Yaskawa INFORM job: SKRZYNIA_5340_0_STOPNI_2OBR.JBI

/JOB
//NAME SKRZYNIA_5340_0_STOPNI_2OBR
///FOLDERNAME 02-SKRZYNIE_JOBS
//POS
///NPOS 607,607,0,50,0,0
///TOOL 0
///POSTYPE PULSE
///PULSE
C00000=1055,-24125,84372,288,19725,204
C00001=0,-15438,65714,0,-68532,0
C00002=4718,-16587,59952,3396,-65485,-935
C00003=32997,-21499,42555,27623,-61436,21376
C00004=31759,-20688,42932,26837,-60850,21559
C00005=28987,-21156,42712,24818,-60442,22222
C00006=33447,-21964,42352,27886,-61721,21330
C00007=37687,-23357,41794,30651,-63289,20620
C00008=38979,-19018,48057,32961,-64962,20678
C00009=37261,-18075,48526,31902,-64209,20901
C00010=35830,-17198,48994,31015,-63571,21092
C00011=34080,-17614,48768,29780,-63290,21485
C00012=37261,-18075,48526,31902,-64209,20901
C00013=47373,-21912,40596,41149,-66086,26950
C00014=45033,-20851,41104,39798,-65001,27223
C00015=42790,-19693,41704,38494,-63946,27495
C00016=41070,-20182,41442,37324,-63566,27891
C00017=45033,-20851,41104,39798,-65001,27223
C00018=45033,-20851,41104,39798,-65001,27223
C00019=59624,-29540,14278,64846,-60867,16042
C00020=57357,-28542,14780,63940,-59509,16120
C00021=56188,-29140,14476,63237,-58995,16387
C00022=59588,-29370,14363,64862,-60819,16012
C00023=62924,-29779,15793,65870,-63073,16252
C00024=59724,-28781,16276,64511,-61238,16415
C00025=57764,-27936,16704,63709,-60078,16488
C00026=56408,-28589,16373,62897,-59486,16787
C00027=59724,-28781,16276,64511,-61238,16415
C00028=87562,-48087,-13810,78020,-75252,11220
C00029=10104,-46603,4759,11228,-37390,-5046
C00030=0,-52280,40443,0,6876,0
C00031=1529,-42140,58025,-5964,2417,3265
C00032=0,-38374,23626,-1605,-51738,268
C00033=45044,-23015,37260,35797,-71879,25522
C00034=39973,-29571,18873,35060,-63052,24165
C00035=38620,-28701,19269,34339,-62304,24363
C00036=36409,-29254,19014,32896,-61805,24958
C00037=44451,-29039,21934,37281,-65892,23702
C00038=49472,-39353,6917,53118,-50908,20251
C00039=45058,-39356,3832,51653,-47640,20099
C00040=42883,-38319,4163,50577,-46309,20295
C00041=40255,-38926,3967,48502,-45334,21060
C00042=46774,-39679,3737,52663,-48537,19827
C00043=48708,-40455,3517,53615,-49689,19657
C00044=43798,-39237,3871,50850,-47027,20335
C00045=41951,-38324,4161,49930,-45891,20507
C00046=39836,-38844,3994,48234,-45126,21137
C00047=48489,-40338,3551,53521,-49551,19665
C00048=48489,-40338,3551,53521,-49551,19665
C00049=44432,-39026,3936,51363,-47247,20139
C00050=42487,-38069,4248,50403,-46050,20315
C00051=39061,-38795,4009,47695,-44769,21310
C00052=44432,-39026,3936,51363,-47247,20139
C00053=45358,-49480,-3557,50155,-49322,21260
C00054=1817,-44984,2816,-3462,-45659,1296
C00055=1445,-28771,30219,-502,-63201,-220
C00056=1148,-56354,34370,-22,3827,-10
C00057=0,-52280,40443,0,6876,0
C00058=0,-49898,44897,0,-65513,0
C00059=52002,-27630,35066,40617,-70496,28619
C00060=38179,-24916,32897,32855,-63545,30206
C00061=36484,-23889,33369,31863,-62698,30449
C00062=33804,-24434,33113,30025,-62179,31112
C00063=38179,-24916,32897,32855,-63545,30206
C00064=78369,-41260,16071,67181,-65880,21417
C00065=137,-45861,52341,97,-67596,-14
C00066=-31499,-58302,-23356,15027,12889,-13082
C00067=-52768,-43016,-26078,18373,38595,-18774
C00068=-89470,-32103,-32973,29905,69139,-31512
C00069=-68838,-26884,-24872,16972,64732,-23076
C00070=-53036,-11528,-12218,12363,64665,-17409
C00071=-51536,-9474,-10276,11905,64649,-16876
C00072=-51739,-9114,-7787,12104,63269,-17104
C00073=-53036,-11528,-12218,12363,64665,-17409
C00074=-17541,-26226,-24397,927,59032,-5038
C00075=-17541,-26226,-24397,927,59032,-5038
C00076=-16950,-23991,-22741,715,59568,-4818
C00077=-17036,-23563,-20101,755,58071,-4857
C00078=-17541,-26226,-24397,927,59032,-5038
C00079=34102,-23192,-21614,-15638,64271,13209
C00080=33423,-21885,-20599,-15423,64418,12942
C00081=32426,-19856,-18975,-15106,64629,12551
C00082=32578,-19611,-17013,-15290,63535,12762
C00083=33423,-21885,-20599,-15423,64418,12942
C00084=59339,-6070,-6417,-20979,72191,20891
C00085=59339,-6070,-6417,-20979,72191,20891
C00086=57897,-4256,-4562,-20702,71913,20431
C00087=58108,-3992,-2506,-20878,70835,20713
C00088=59339,-6070,-6417,-20979,72191,20891
C00089=42744,-35904,-30225,-18322,62562,16651
C00090=-53036,-11528,-12218,12363,64665,-17409
C00091=-77982,-26538,-29134,27151,66629,-27745
C00092=-70983,-8594,-1966,26503,59809,-49670
C00093=-80152,19776,40785,37351,72704,-50428
C00094=-79984,20154,42529,37516,71911,-50638
C00095=-79233,18397,40079,37458,71885,-50340
C00096=-79984,20154,42529,37516,71911,-50638
C00097=-73519,23289,38838,28890,77081,-45618
C00098=-73519,24511,42682,29072,75582,-46027
C00099=-73519,23289,38838,28890,77081,-45618
C00100=-88897,15706,42282,50101,71325,-56974
C00101=-88897,15706,42282,50101,71325,-56974
C00102=-87612,12343,37838,50071,70996,-56519
C00103=-85283,14202,40272,50301,69633,-56165
C00104=-87338,12550,38107,50098,70839,-56476
C00105=-84952,-1789,13569,34660,47724,-58955
C00106=-67641,-1674,11109,10330,44856,-44725
C00107=-66443,961,13975,9688,44721,-44210
C00108=-67641,-1674,11109,10330,44856,-44725
C00109=-67641,-376,15347,10694,42950,-44967
C00110=-67641,-1674,11109,10330,44856,-44725
C00111=-79040,417,20398,15965,28992,-57786
C00112=-76655,5212,30978,15501,25024,-57306
C00113=-76655,6949,35816,16758,23084,-57955
C00114=-76655,5212,30978,15501,25024,-57306
C00115=-74761,6919,33010,13466,24593,-56049
C00116=-80460,-2874,12270,15804,32253,-57809
C00117=-61258,-29124,-13156,26560,43617,-22150
C00118=-30420,-40507,-29240,27153,53235,15188
C00119=-18589,-38725,-21450,23338,47896,18931
C00120=-17722,-35233,-16455,23322,46926,19051
C00121=-17722,-33749,-12435,23948,45421,18620
C00122=-17722,-33892,-12819,23887,45564,18661
C00123=-16677,-31133,-11209,23138,46167,19311
C00124=-17819,-35820,-17540,23246,47228,19090
C00125=-74104,-11494,-6266,31916,75042,4269
C00126=-71226,-7329,2631,32115,71468,4273
C00127=-71226,-6504,5446,32343,70365,3922
C00128=-71226,-6611,5086,32313,70505,3967
C00129=-68386,-4058,7675,32040,69573,4789
C00130=-73314,-9412,-353,32206,72648,3829
C00131=51751,-31069,-22965,-10739,49070,48663
C00132=49028,-23852,-11575,-9841,46366,47823
C00133=49028,-23004,-8935,-10039,45204,47956
C00134=49028,-23118,-9286,-10013,45357,47939
C00135=47000,-20813,-7527,-8928,45644,47024
C00136=50476,-26208,-15307,-10408,47325,48332
C00137=90602,-5375,6902,-38786,69848,59444
C00138=83174,19950,50269,-44999,67580,58220
C00139=82362,17902,47383,-44926,67511,57879
C00140=83515,19072,48341,-44798,68200,58056
C00141=78091,19382,40247,-36371,72286,52960
C00142=78091,20664,44011,-36670,70997,53443
C00143=78091,19382,40247,-36371,72286,52960
C00144=88699,7296,38566,-55615,63182,60372
C00145=86803,3068,32674,-55410,62638,59657
C00146=84852,4315,34115,-55564,61561,59330
C00147=86803,3068,32674,-55410,62638,59657
C00148=92770,-2803,21719,-53893,67577,59421
C00149=73393,-10627,10934,-27897,30744,62458
C00150=70789,-6606,18800,-27824,27830,62140
C00151=69654,-4593,20814,-26755,27596,61444
C00152=70789,-6606,18800,-27824,27830,62140
C00153=70789,-5070,23059,-29482,26284,63017
C00154=70789,-6606,18800,-27824,27830,62140
C00155=83486,-8736,6503,-27040,35338,66550
C00156=77831,-2041,26192,-25270,18452,68895
C00157=77967,1961,32070,-26860,17569,69698
C00158=77967,5243,40752,-32914,14549,72656
C00159=77967,1961,32070,-26860,17569,69698
C00160=74560,4730,35257,-21622,16551,66717
C00161=77967,1961,32070,-26860,17569,69698
C00162=81109,-22356,2664,-22493,33121,60116
C00163=86168,-49730,-13668,-23926,46819,49343
C00164=44183,-52048,-7537,-24795,46064,51426
C00165=0,-52280,40443,0,6876,0
C00166=0,-52280,40443,0,6876,0
C00167=33629,-57276,-6399,46271,-24969,-2804
C00168=75493,-63502,-64712,103874,-64610,-6298
C00169=47446,-58597,-62761,109790,-45856,-10712
C00170=43673,-60069,-65334,114064,-43025,-9215
C00171=55379,-67378,-68041,108237,-48773,-4935
C00172=62671,-64213,-64640,104431,-56093,-7372
C00173=28458,-50318,6850,47420,-25887,-3347
C00174=0,-52280,40443,0,6876,0
C00175=1055,-24125,84372,288,19725,204
C00176=0,-15438,65714,0,-68532,0
C00177=0,-15438,65714,966,-70097,42926
C00178=69988,-9219,57065,61610,-82752,27767
C00179=63113,-6157,59685,58080,-79692,28271
C00180=46309,-5455,68070,40267,-75151,29719
C00181=49471,-5188,67710,43421,-76082,29577
C00182=63113,-6157,59685,58080,-79692,28271
C00183=69988,-9219,57065,61610,-82752,27767
C00184=0,-15438,65714,966,-70097,42926
C00185=0,-15438,65714,0,-68532,0
C00186=1055,-24125,84372,288,19725,204
C00187=1055,-24125,84372,288,19725,204
C00188=0,-52280,40443,0,6876,0
C00189=0,-17525,61946,0,273,32004
C00190=54446,-4421,37881,-48560,57645,57448
C00191=45059,-5790,38757,-53071,45868,54447
C00192=47306,-4859,57027,-85859,41058,71744
C00193=46362,-329,57203,-69834,42671,59860
C00194=35194,-2896,34959,-39493,48020,38101
C00195=43067,2853,36106,-38598,60324,43004
C00196=45059,-5790,38757,-53071,45868,54447
C00197=54446,-4421,37881,-48560,57645,57448
C00198=0,-17525,61946,0,273,32004
C00199=0,-52280,40443,0,6876,0
C00200=0,-52280,40443,0,6876,0
C00201=0,-52280,40443,0,6876,0
C00202=0,-52280,40443,0,-42737,40640
C00203=0,-52280,40443,0,-42737,40640
C00204=64551,-35409,28076,75550,-44539,17239
C00205=49799,-25338,45366,61341,-39751,21495
C00206=45731,-22710,35392,68644,-36821,18294
C00207=38151,-27944,23982,59630,-35957,20215
C00208=38219,-25330,29845,57337,-37014,21581
C00209=43117,-27612,29118,67655,-35359,18183
C00210=39863,-22026,47404,54615,-35502,22403
C00211=0,-52277,40442,0,6872,2
C00212=0,-38538,66749,0,-898,0
C00213=0,-52280,40443,0,-79033,35417
C00214=46775,-35113,22190,42926,-67531,20697
C00215=52587,-26056,25345,47610,-66542,17970
C00216=46075,-25504,24484,44216,-63256,18807
C00217=46254,-27712,19552,44922,-62123,18131
C00218=53914,-29436,22058,48262,-67266,17843
C00219=46775,-35113,22190,42926,-67531,20697
C00220=0,-52280,40443,0,-79033,35417
C00221=0,-52280,40443,0,-61239,28081
C00222=53819,-14110,13758,-46164,60155,50576
C00223=48398,-14119,9451,-44868,59619,48162
C00224=41013,-18640,20407,-60592,39621,52880
C00225=26504,-16872,16016,-34457,37392,33859
C00226=48398,-14119,9451,-44868,59619,48162
C00227=53819,-14110,13758,-46164,60155,50576
C00228=0,-52280,40443,0,-61239,28081
C00229=404,-42897,57020,-1574,2523,869
C00230=404,-42897,57020,-1574,2523,869
C00231=0,-52280,40443,0,6876,0
C00232=-99253,-13690,44082,59847,13407,-31313
C00233=-87814,-12734,20141,45739,-14352,-64418
C00234=-86669,-6582,30812,41148,-16781,-62025
C00235=-85055,-5827,31548,44003,-17420,-63187
C00236=-85971,-6262,31124,42409,-17052,-62539
C00237=-86650,-5303,32069,41395,-16716,-62141
C00238=-94954,-14494,-1860,-7818,15857,-59130
C00239=-94513,13660,61459,-3970,3134,-58997
C00240=-94981,20459,77123,-7495,-2517,-57346
C00241=-85971,-6262,31124,42409,-17052,-62539
C00242=-86125,-12470,22545,29004,-25567,-58412
C00243=-83883,-11340,22525,32952,-25567,-60136
C00244=-82768,-10824,22986,34487,-25904,-60776
C00245=-83883,-11340,22525,32952,-25567,-60136
C00246=-85143,-9772,23941,31487,-24966,-59556
C00247=-83883,-11340,22525,32952,-25567,-60136
C00248=-85732,-21202,11427,30682,-24763,-59235
C00249=-84150,-10929,23786,31981,-25941,-59678
C00250=-83036,-10419,24246,33504,-26268,-60308
C00251=-84150,-10929,23786,31981,-25941,-59678
C00252=-85291,-9507,25078,30650,-25411,-59154
C00253=-84150,-10929,23786,31981,-25941,-59678
C00254=-85786,-16909,14677,31743,-23900,-59790
C00255=-84150,-10498,24888,31517,-26306,-59436
C00256=-83174,-10052,25293,32841,-26587,-59984
C00257=-84150,-10498,24888,31517,-26306,-59436
C00258=-85258,-9112,26156,30226,-25800,-58928
C00259=-84150,-10498,24888,31517,-26306,-59436
C00260=-87841,-18519,13420,28367,-23534,-58339
C00261=-85040,-10859,24618,30253,-26091,-58908
C00262=-83241,-10052,25348,32714,-26598,-59924
C00263=-84150,-10465,24972,31484,-26336,-59417
C00264=-85145,-9228,26102,30329,-25881,-58963
C00265=-84150,-10465,24972,31484,-26336,-59417
C00266=-86371,-18277,13606,30568,-23951,-59265
C00267=-84345,-11688,21985,32461,-25312,-59957
C00268=-83211,-11173,22442,34044,-25650,-60618
C00269=-84345,-11688,21985,32461,-25312,-59957
C00270=-85283,-10526,23025,31366,-24861,-59525
C00271=-84345,-11688,21985,32461,-25312,-59957
C00272=-86191,-19647,12567,30467,-24278,-59187
C00273=-84345,-10877,24073,31552,-26006,-59481
C00274=-83051,-10286,24607,33321,-26381,-60213
C00275=-84345,-10877,24073,31552,-26006,-59481
C00276=-85179,-9842,25009,30582,-25619,-59100
C00277=-84345,-10877,24073,31552,-26006,-59481
C00278=-85438,-18022,14839,31140,-24818,-59429
C00279=-84247,-11820,22550,32049,-25753,-59727
C00280=-84104,-10976,23642,32111,-25899,-59738
C00281=-82990,-10465,24105,33639,-26227,-60372
C00282=-84104,-10976,23642,32111,-25899,-59738
C00283=-84898,-9998,24525,31196,-25529,-59378
C00284=-84104,-10976,23642,32111,-25899,-59738
C00285=-86610,-16845,14732,30573,-23614,-59301
C00286=-84104,-10864,23927,31990,-25993,-59674
C00287=-82824,-10273,24459,33737,-26370,-60397
C00288=-84104,-10864,23927,31990,-25993,-59674
C00289=-84789,-10021,24690,31200,-25673,-59363
C00290=-84104,-10864,23927,31990,-25993,-59674
C00291=-83806,-19585,12613,33764,-25080,-60559
C00292=-83924,-10205,25475,31619,-26533,-59453
C00293=-82780,-9675,25960,33156,-26866,-60087
C00294=-83924,-10205,25475,31619,-26533,-59453
C00295=-84478,-9530,26093,30986,-26280,-59206
C00296=-83924,-10205,25475,31619,-26533,-59453
C00297=-87149,-17993,13826,29513,-23647,-58830
C00298=-84920,-13182,20975,31162,-25481,-59361
C00299=-83711,-10572,24852,32056,-26475,-59649
C00300=-82779,-10142,25241,33309,-26748,-60166
C00301=-83711,-10572,24852,32056,-26475,-59649
C00302=-84370,-9774,25579,31305,-26170,-59356
C00303=-83711,-10572,24852,32056,-26475,-59649
C00304=-83642,-3679,42021,23358,-36761,-56118
C00305=-85886,-5975,41264,18964,-40261,-54782
C00306=-83919,-11632,22322,32811,-25616,-60079
C00307=-82884,-11162,22742,34234,-25925,-60671
C00308=-83919,-11632,22322,32811,-25616,-60079
C00309=-84723,-10654,23196,31887,-25230,-59715
C00310=-83919,-11632,22322,32811,-25616,-60079
C00311=-87348,-16035,7353,17528,-35245,-56477
C00312=-86244,-15062,8172,18754,-35315,-57058
C00313=-86244,-16649,3638,19674,-33501,-57585
C00314=-85308,-16228,3988,20718,-33648,-58082
C00315=-86244,-16649,3638,19674,-33501,-57585
C00316=-86740,-15973,4201,19194,-33277,-57362
C00317=-86244,-16649,3638,19674,-33501,-57585
C00318=-73780,-8639,20128,34258,-51705,-52097
C00319=-90711,-17528,-28778,11328,-28245,-57111
C00320=-92565,-19610,-33223,7138,-24591,-57051
C00321=-91512,-19116,-32812,8551,-24603,-57834
C00322=-92565,-19610,-33223,7138,-24591,-57051
C00323=-93003,-18716,-32476,6600,-24397,-56752
C00324=-92565,-19610,-33223,7138,-24591,-57051
C00325=-92565,-19610,-33223,7138,-24591,-57051
C00326=-95836,-54375,-51122,6031,-17685,-48210
C00327=-95836,-54375,-51122,6031,-17685,-48210
C00328=-43821,-47238,-2775,-3022,56549,-3681
C00329=-20126,-26882,59542,2406,16879,-9162
C00330=-20126,-26882,59542,2406,16879,-9162
C00331=98601,-10520,92678,4674,-40855,-9615
C00332=95537,-19831,-2695,-2933,-44471,35837
C00333=92548,-20391,-28429,-6186,-30623,55200
C00334=91429,-17018,-28974,-8057,-27827,56250
C00335=91429,-17018,-28974,-8057,-27827,56250
C00336=90371,-16495,-28521,-9286,-27856,56953
C00337=91429,-17018,-28974,-8057,-27827,56250
C00338=92033,-15799,-27911,-7415,-27588,55880
C00339=91429,-17018,-28974,-8057,-27827,56250
C00340=92548,-20391,-28429,-6186,-30623,55200
C00341=91156,-15018,-4648,-8036,-38181,54813
C00342=90585,-14766,-4428,-8565,-38201,55100
C00343=88830,-13959,-3717,-10186,-38284,55977
C00344=89897,-14456,-4157,-9202,-38230,55445
C00345=90761,-12944,-2809,-8452,-37927,55043
C00346=89897,-14456,-4157,-9202,-38230,55445
C00347=89910,-11217,67535,-9455,-58896,55399
C00348=89910,-11217,67535,-9455,-58896,55399
C00349=85786,-16735,14816,-31782,-23869,59812
C00350=83514,-12996,17929,-35760,-24132,61552
C00351=82251,-12406,18443,-37550,-24551,62308
C00352=83514,-12996,17929,-35760,-24132,61552
C00353=84258,-12095,18717,-34917,-23742,61217
C00354=83514,-12996,17929,-35760,-24132,61552
C00355=87149,-17993,13826,-29513,-23647,58830
C00356=83118,-12818,18089,-36330,-24263,61791
C00357=81915,-12248,18589,-38020,-24666,62504
C00358=83118,-12818,18089,-36330,-24263,61791
C00359=83897,-11882,18912,-35460,-23856,61445
C00360=83118,-12818,18089,-36330,-24263,61791
C00361=83806,-19585,12613,-33764,-25080,60559
C00362=82998,-13006,17925,-36445,-24332,61826
C00363=81675,-12378,18472,-38297,-24777,62607
C00364=82998,-13006,17925,-36445,-24332,61826
C00365=83876,-11958,18841,-35466,-23874,61442
C00366=82998,-13006,17925,-36445,-24332,61826
C00367=86610,-16845,14732,-30573,-23614,59301
C00368=82493,-13239,17725,-37070,-24559,62089
C00369=81406,-12724,18174,-38578,-24928,62723
C00370=82493,-13239,17725,-37070,-24559,62089
C00371=83436,-12134,18690,-36041,-24064,61684
C00372=82493,-13239,17725,-37070,-24559,62089
C00373=84814,-16043,15376,-33312,-24093,60464
C00374=82555,-13613,17404,-36910,-24580,62015
C00375=81384,-13062,17878,-38534,-24974,62698
C00376=82555,-13613,17404,-36910,-24580,62015
C00377=83566,-12434,18427,-35805,-24047,61580
C00378=82555,-13613,17404,-36910,-24580,62015
C00379=86191,-19647,12567,-30467,-24278,59187
C00380=82500,-13648,17375,-36975,-24607,62039
C00381=81467,-13161,17792,-38413,-24955,62645
C00382=82500,-13648,17375,-36975,-24607,62039
C00383=83481,-12505,18364,-35905,-24087,61617
C00384=82500,-13648,17375,-36975,-24607,62039
C00385=86371,-18277,13606,-30568,-23951,59265
C00386=82904,-13790,17251,-36416,-24470,61808
C00387=81715,-13237,17726,-38081,-24865,62509
C00388=82904,-13790,17251,-36416,-24470,61808
C00389=83686,-12878,18037,-35556,-24055,61469
C00390=82904,-13790,17251,-36416,-24470,61808
C00391=87841,-18519,13420,-28367,-23534,58339
C00392=82748,-13879,17174,-36603,-24542,61883
C00393=81692,-13388,17594,-38077,-24893,62505
C00394=82748,-13879,17174,-36603,-24542,61883
C00395=83607,-12881,18032,-35663,-24082,61515
C00396=82748,-13879,17174,-36603,-24542,61883
C00397=85786,-16909,14677,-31743,-23900,59790
C00398=82520,-14198,16902,-36833,-24674,61972
C00399=81460,-13708,17319,-38301,-25026,62591
C00400=82520,-14198,16902,-36833,-24674,61972
C00401=83571,-12989,17938,-35691,-24113,61524
C00402=82520,-14198,16902,-36833,-24674,61972
C00403=85732,-21202,11427,-30682,-24763,59235
C00404=82398,-14365,16763,-36952,-24745,62014
C00405=81172,-13798,17245,-38643,-25153,62725
C00406=82398,-14365,16763,-36952,-24745,62014
C00407=83600,-12984,17944,-35650,-24102,61504
C00408=82398,-14365,16763,-36952,-24745,62014
C00409=92346,-18713,13565,-21110,-22545,55257
C00410=82794,-13980,17083,-36511,-24538,61844
C00411=81518,-13384,17592,-38292,-24965,62594
C00412=82794,-13980,17083,-36511,-24538,61844
C00413=83714,-12912,18003,-35501,-24048,61445
C00414=82794,-13980,17083,-36511,-24538,61844
C00415=86140,-12802,12665,-93523,-10743,85795
C00416=86140,-12802,12665,-93523,-10743,85795
C00417=85030,-12289,13120,-93723,-11463,85776
C00418=86140,-12802,12665,-93523,-10743,85795
C00419=86958,-11660,13681,-94506,-10238,86349
C00420=86140,-12802,12665,-93523,-10743,85795
C00421=86625,-13020,12474,-93432,-10428,85802
C00422=86720,-13063,12436,-93414,-10366,85804
C00423=85672,-12588,12853,-93609,-11048,85787
C00424=86091,-12781,12683,-93534,-10775,85794
C00425=86978,-11540,13790,-94601,-10225,86395
C00426=86091,-12781,12683,-93534,-10775,85794
C00427=86674,107,23869,25042,24033,51593
C00428=86674,107,23869,25042,24033,51593
C00429=86674,1750,28532,27061,22272,50559
C00430=86674,107,23869,25042,24033,51593
C00431=86830,-21199,-17039,14859,33768,55796
C00432=85045,-36869,-4353,-28502,-22832,52282
C00433=0,-24029,84339,0,19981,0
C00434=0,-24029,84339,0,19981,0
C00435=3172,-24246,80980,3465,15913,689
C00436=-86563,-26985,13879,10257,-21548,-45530
C00437=-86191,-19647,12567,30467,-24278,-59187
C00438=-83221,-13587,17636,37793,-25116,-62228
C00439=-91978,-13833,14560,12391,-18633,-51524
C00440=-94992,-13830,14285,1276,-18012,-46664
C00441=-84074,-17488,11256,38660,-23649,-62784
C00442=-73679,-33270,1000,44272,-31600,-64253
C00443=-86926,-60758,23267,6576,1160,-9545
C00444=0,-52280,40443,0,6876,0
C00445=82475,-58079,26734,835,4084,4444
C00446=97932,-26840,7691,8784,-23444,42538
C00447=87166,-16607,16322,-25365,-24201,56345
C00448=84699,-11354,21752,-29145,-24735,57949
C00449=84804,-11023,22730,-28561,-25071,57659
C00450=85100,-26994,10417,-24982,-28140,55821
C00451=0,-52280,40443,0,6876,0
C00452=0,-52280,40443,0,6876,0
C00453=-90140,-60305,18108,-2708,1721,-7625
C00454=-95594,-27428,6866,-4663,-19832,-42154
C00455=-98688,-13767,16447,-18366,-10080,-35766
C00456=-98964,-4977,31041,-27811,-8682,-30400
C00457=-98987,-3006,34487,-29035,-8628,-29652
C00458=-99668,3923,47993,-36046,-8554,-25749
C00459=-97898,6199,51529,-29419,-5862,-29460
C00460=-93331,7027,46084,-21637,6926,-34654
C00461=-93331,9643,52589,-32935,4701,-29330
C00462=-91881,12566,59903,-8075,11651,-42601
C00463=-91392,18044,70719,-12774,8436,-40275
C00464=-95084,15513,53253,-335,18313,-46866
C00465=-99268,-13088,27343,-18620,-14105,-35021
C00466=-90140,-60305,18108,-2708,1721,-7625
C00467=0,-52280,40443,0,6876,0
C00468=84259,-57935,27522,-3761,3673,6310
C00469=86507,-39672,4297,-27618,-16640,46340
C00470=73669,-37119,-20783,-92053,-19719,85232
C00471=86539,-20830,1725,-71850,-11773,76853
C00472=94927,-16191,10904,-46169,-1414,61414
C00473=97704,-11547,13178,-56709,4181,66931
C00474=98708,-8628,11747,-16202,14842,48818
C00475=96432,-319,21323,-3495,24089,38404
C00476=97976,685,17732,-6153,31139,39163
C00477=96085,-4775,15361,-2075,25096,37900
C00478=101780,15887,17889,-10773,66834,38316
C00479=97846,5957,18050,-4866,41853,38411
C00480=100487,-9453,-1206,-10413,41328,41147
C00481=96250,-19428,-8283,-4838,27297,37910
C00482=86507,-39672,4297,-27618,-16640,46340
C00483=84259,-57935,27522,-3761,3673,6310
C00484=0,-52280,40443,0,6876,0
C00485=0,-27933,77061,0,20812,0
C00486=0,-27933,77061,0,20812,0
C00487=0,-52280,40443,0,6876,0
C00488=-91970,-60791,14435,-3343,512,-9412
C00489=-98647,-24138,10005,-11519,-21203,-39749
C00490=-99883,-13980,22886,-11640,-25090,-40341
C00491=-99702,-9154,61728,-1148,-61809,-40243
C00492=-84328,-13042,29707,23458,-33731,-54641
C00493=-83101,-4179,39208,25894,-34785,-55667
C00494=-82881,-4330,38692,26392,-34479,-55866
C00495=-76259,-18287,26646,31659,-38322,-57579
C00496=-89741,-28009,12101,4461,-28076,-46404
C00497=-91970,-60791,14435,-3343,512,-9412
C00498=0,-52280,40443,0,6876,0
C00499=91083,-60784,14823,-9043,-825,15173
C00500=83869,-19403,12921,-33769,-24740,60260
C00501=83869,-19403,12921,-33769,-24740,60260
C00502=83932,-19538,53415,-33663,-71112,60249
C00503=83932,-19538,53415,-33663,-71112,60249
C00504=82480,-12247,21118,-35440,-26416,60009
C00505=82194,-11433,19802,-37650,-25323,61125
C00506=81904,-9374,24711,-35791,-26879,60109
C00507=79790,-20261,14917,-36681,-28829,60258
C00508=76554,-29711,-1870,-46042,-25952,65654
C00509=91083,-60784,14823,-9043,-825,15173
C00510=0,-52280,40443,0,6876,0
C00511=-91526,-60598,16699,7584,176,-13289
C00512=-81382,-25890,9219,35455,-25500,-59095
C00513=-86453,-20958,12525,30076,-22568,-57089
C00514=-86589,-16097,16237,31250,-21582,-57704
C00515=-98933,-11298,20505,-13970,-18736,-37953
C00516=-98281,-10965,21163,-11559,-18548,-39330
C00517=-85424,-18472,14402,34409,-22969,-58895
C00518=-74746,-27148,8488,44263,-29128,-62418
C00519=-81326,-27507,8265,35533,-26282,-59001
C00520=-91415,-60262,16631,7870,-73,-13734
C00521=24,-24029,84339,7,19981,5
C00522=100404,-52373,45687,-1822,14816,-5144
C00523=75939,-26469,7919,-40869,-29645,63133
C00524=81882,-22565,10470,-35355,-26404,61107
C00525=82801,-12246,21732,-34208,-26055,60642
C00526=91844,-10818,23389,-8611,-22226,49798
C00527=96558,-9677,26191,5829,-23135,43648
C00528=77262,-23244,14300,-38922,-31295,61912
C00529=78410,-22868,15324,-38001,-30064,61274
C00530=96357,-33562,33410,58602,-23427,10353
C00531=568,-24029,84339,168,19981,112
C00532=-91970,-60791,14435,-3343,512,-9412
C00533=-98991,-22833,11519,-12824,-17638,-36336
C00534=-86376,-13627,18436,38326,-18406,-58533
C00535=-85581,-10814,20279,41280,-18093,-59893
C00536=-85551,-10406,21021,40925,-18257,-59713
C00537=-86274,-24518,9978,34497,-20333,-56613
C00538=-91684,-53777,2301,20525,-9313,-33684
C00539=-67305,-55044,34987,1504,5690,-2468
C00540=0,-52280,40443,0,6876,0
C00541=77036,-56616,31288,-2531,4707,4197
C00542=84359,-28321,8817,-32860,-20485,54199
C00543=81156,-16932,14874,-39538,-26422,62851
C00544=93122,-15135,13007,-5735,-18111,48773
C00545=90767,-14192,15510,-13532,-19632,52035
C00546=77970,-27630,4721,-41834,-28549,63607
C00547=81111,-35571,7141,-33980,-21909,52006
C00548=82626,-57814,28323,-4146,3364,6346
C00549=0,-52280,40443,0,6876,0
C00550=0,-28135,76691,0,20839,0
C00551=0,-28135,76691,0,20839,0
C00552=-45332,-39712,59352,-1730,18713,2903
C00553=-94065,-8316,59352,-1730,-37754,-40387
C00554=-100331,-14895,33931,-8215,-36518,-40227
C00555=-98931,-8578,39429,-6260,-48307,-43744
C00556=-100336,-4176,46216,-7600,-55875,-44633
C00557=-93952,8947,73671,995,-68520,-43850
C00558=-98791,-3170,32594,-4861,-60761,-43748
C00559=-98768,4156,37660,-4945,-58738,-43661
C00560=-98673,-12696,-17797,-7569,-33360,-41896
C00561=-99330,-14840,-29426,-9917,-27109,-40593
C00562=-99605,-15546,-21493,-8548,-33053,-41326
C00563=-100467,-8208,-2562,-8095,-44661,-42156
C00564=-93952,8947,73671,995,-68520,-43850
C00565=-88754,54,62805,4404,-67858,-45120
C00566=-100222,-4532,45667,-7492,-55263,-44561
C00567=-100331,-14895,33931,-8215,-36518,-40227
C00568=-94065,-8316,59352,-1730,-37754,-40387
C00569=-45544,-32973,71870,-2133,15168,3033
C00570=0,-28135,76691,0,20839,0
C00571=54178,-17846,77779,596,-29686,20997
C00572=54178,-17846,77779,596,-29686,20997
C00573=99462,-18987,75418,611,-28919,20989
C00574=98707,-9390,78674,1080,-71212,38250
C00575=98768,-5182,41096,1808,-44974,38308
C00576=100431,1771,51615,3823,-56746,39115
C00577=97953,-6621,17555,2289,-50176,39420
C00578=95834,-5353,18817,760,-50052,40242
C00579=86453,-3910,18511,-13431,-48443,44868
C00580=88887,-11110,-8515,-11527,-36861,46615
C00581=88808,-13839,-20865,-13699,-30585,47852
C00582=90457,-16080,-12990,-9972,-37305,45724
C00583=97953,-6621,17555,2289,-50176,39420
C00584=100431,1771,51615,3823,-56746,39115
C00585=98768,-5182,41096,1808,-44974,38308
C00586=98707,-9390,78674,1080,-71212,38250
C00587=0,-28135,76691,0,20839,0
C00588=0,-28135,76691,0,20839,0
C00589=-91526,-60598,16699,7584,176,-13289
C00590=-81382,-25890,9219,35455,-25500,-59095
C00591=-81382,-25890,9219,35455,-25500,-59095
C00592=-85509,-13950,19358,32213,-22393,-58041
C00593=-96341,-12086,19487,-5053,-17846,-42145
C00594=-97523,-9822,24708,-8570,-19966,-40659
C00595=-84656,-25369,12054,31249,-26195,-57129
C00596=-82652,-57346,29982,2770,3944,-5064
C00597=0,-52280,40443,0,6876,0
C00598=60653,-54633,35892,-1212,5841,2035
C00599=77942,-28227,6869,-38010,-29303,61907
C00600=82500,-13648,17375,-36975,-24607,62039
C00601=80731,-11587,18684,-41654,-25449,63953
C00602=80409,-10373,22284,-40214,-26848,63104
C00603=64389,-31987,5108,-50419,-37074,66126
C00604=60653,-54633,35892,-1212,5841,2035
C00605=0,-52280,40443,0,6876,0
C00606=0,-28167,76633,0,20843,0
BC00000=413138
BC00001=413138
BC00002=388163
BC00003=356740
BC00004=356740
BC00005=356740
BC00006=356740
BC00007=356740
BC00008=407176
BC00009=407176
BC00010=407176
BC00011=407176
BC00012=407176
BC00013=479433
BC00014=479433
BC00015=479433
BC00016=479433
BC00017=479433
BC00018=530237
BC00019=530237
BC00020=530237
BC00021=530237
BC00022=530237
BC00023=601977
BC00024=601977
BC00025=601977
BC00026=601977
BC00027=601977
BC00028=601977
BC00029=522422
BC00030=522422
BC00031=671734
BC00032=689202
BC00033=689202
BC00034=689202
BC00035=689202
BC00036=689202
BC00037=689202
BC00038=726463
BC00039=726463
BC00040=726463
BC00041=726463
BC00042=726463
BC00043=782137
BC00044=782137
BC00045=782137
BC00046=782137
BC00047=782137
BC00048=850421
BC00049=850421
BC00050=850421
BC00051=850421
BC00052=850421
BC00053=850421
BC00054=823841
BC00055=797607
BC00056=755227
BC00057=755227
BC00058=915219
BC00059=914226
BC00060=914226
BC00061=914226
BC00062=914226
BC00063=914226
BC00064=914226
BC00065=922367
BC00066=927819
BC00067=927819
BC00068=927819
BC00069=943180
BC00070=943180
BC00071=943180
BC00072=943180
BC00073=943180
BC00074=943180
BC00075=943180
BC00076=943180
BC00077=943180
BC00078=943180
BC00079=943180
BC00080=943180
BC00081=943180
BC00082=943180
BC00083=943180
BC00084=943180
BC00085=943180
BC00086=943180
BC00087=943180
BC00088=943180
BC00089=943180
BC00090=943180
BC00091=943180
BC00092=943180
BC00093=943180
BC00094=943182
BC00095=943182
BC00096=943182
BC00097=943182
BC00098=943182
BC00099=943182
BC00100=943182
BC00101=943182
BC00102=943182
BC00103=943182
BC00104=943182
BC00105=943182
BC00106=943182
BC00107=943182
BC00108=943182
BC00109=943182
BC00110=943182
BC00111=943182
BC00112=943182
BC00113=943182
BC00114=943182
BC00115=943182
BC00116=943182
BC00117=943183
BC00118=943184
BC00119=943184
BC00120=943184
BC00121=943184
BC00122=943184
BC00123=943184
BC00124=943184
BC00125=943184
BC00126=943184
BC00127=943184
BC00128=943184
BC00129=943156
BC00130=943170
BC00131=943170
BC00132=943170
BC00133=943170
BC00134=943170
BC00135=943170
BC00136=943170
BC00137=943184
BC00138=943184
BC00139=943184
BC00140=943184
BC00141=943184
BC00142=943184
BC00143=943184
BC00144=943184
BC00145=943184
BC00146=943184
BC00147=943184
BC00148=943184
BC00149=943184
BC00150=943184
BC00151=943184
BC00152=943184
BC00153=943184
BC00154=943184
BC00155=943184
BC00156=943184
BC00157=943184
BC00158=943184
BC00159=943184
BC00160=943184
BC00161=943184
BC00162=911399
BC00163=884954
BC00164=838173
BC00165=838173
BC00166=727925
BC00167=734552
BC00168=750834
BC00169=750837
BC00170=810605
BC00171=811927
BC00172=760768
BC00173=744267
BC00174=744267
BC00175=413138
BC00176=413138
BC00177=413138
BC00178=408626
BC00179=408626
BC00180=408753
BC00181=347392
BC00182=408626
BC00183=408626
BC00184=413138
BC00185=413138
BC00186=413138
BC00187=505502
BC00188=697681
BC00189=697681
BC00190=733666
BC00191=758324
BC00192=766520
BC00193=794510
BC00194=817294
BC00195=794510
BC00196=758324
BC00197=733666
BC00198=697681
BC00199=697681
BC00200=697681
BC00201=841681
BC00202=841681
BC00203=884227
BC00204=901088
BC00205=895224
BC00206=896289
BC00207=924873
BC00208=968077
BC00209=921975
BC00210=887634
BC00211=824879
BC00212=507816
BC00213=507816
BC00214=552804
BC00215=552804
BC00216=551170
BC00217=493239
BC00218=491979
BC00219=552804
BC00220=507816
BC00221=507816
BC00222=507816
BC00223=531288
BC00224=531293
BC00225=591068
BC00226=531288
BC00227=507816
BC00228=507816
BC00229=507816
BC00230=737809
BC00231=848972
BC00232=861901
BC00233=963633
BC00234=963633
BC00235=963633
BC00236=963633
BC00237=963633
BC00238=963633
BC00239=963633
BC00240=963633
BC00241=963633
BC00242=963633
BC00243=963633
BC00244=963633
BC00245=963633
BC00246=963633
BC00247=963633
BC00248=902188
BC00249=895372
BC00250=895372
BC00251=895372
BC00252=895372
BC00253=895372
BC00254=840744
BC00255=840744
BC00256=840744
BC00257=840744
BC00258=840744
BC00259=840744
BC00260=779300
BC00261=771332
BC00262=771332
BC00263=771332
BC00264=771332
BC00265=771332
BC00266=717855
BC00267=717855
BC00268=717855
BC00269=717855
BC00270=717855
BC00271=717855
BC00272=656405
BC00273=649173
BC00274=649173
BC00275=649173
BC00276=649173
BC00277=649173
BC00278=594961
BC00279=594961
BC00280=594961
BC00281=594961
BC00282=594961
BC00283=594961
BC00284=594961
BC00285=533517
BC00286=525229
BC00287=525229
BC00288=525229
BC00289=525229
BC00290=525229
BC00291=472073
BC00292=472073
BC00293=472073
BC00294=472073
BC00295=472073
BC00296=472073
BC00297=410629
BC00298=405662
BC00299=402968
BC00300=402968
BC00301=402968
BC00302=402968
BC00303=402968
BC00304=402968
BC00305=349186
BC00306=349186
BC00307=349186
BC00308=349186
BC00309=349186
BC00310=349186
BC00311=336469
BC00312=336469
BC00313=336469
BC00314=336469
BC00315=336469
BC00316=336469
BC00317=336469
BC00318=367602
BC00319=367601
BC00320=367601
BC00321=367601
BC00322=367601
BC00323=367601
BC00324=367601
BC00325=425303
BC00326=425303
BC00327=514953
BC00328=463119
BC00329=419862
BC00330=484962
BC00331=484962
BC00332=395463
BC00333=369502
BC00334=369502
BC00335=369502
BC00336=369502
BC00337=369502
BC00338=369502
BC00339=369502
BC00340=369502
BC00341=368885
BC00342=368885
BC00343=368885
BC00344=368885
BC00345=368885
BC00346=368885
BC00347=419064
BC00348=366918
BC00349=349186
BC00350=353241
BC00351=353241
BC00352=353241
BC00353=353241
BC00354=353241
BC00355=410629
BC00356=409135
BC00357=409135
BC00358=409135
BC00359=409135
BC00360=409135
BC00361=472073
BC00362=476126
BC00363=476126
BC00364=476126
BC00365=476126
BC00366=476126
BC00367=533517
BC00368=532644
BC00369=532644
BC00370=532644
BC00371=532644
BC00372=532644
BC00373=594961
BC00374=599988
BC00375=599988
BC00376=599988
BC00377=599988
BC00378=599988
BC00379=656405
BC00380=653254
BC00381=653254
BC00382=653254
BC00383=653254
BC00384=653254
BC00385=717855
BC00386=721570
BC00387=721570
BC00388=721570
BC00389=721570
BC00390=721570
BC00391=779300
BC00392=777963
BC00393=777963
BC00394=777963
BC00395=777963
BC00396=777963
BC00397=840744
BC00398=843810
BC00399=843810
BC00400=843810
BC00401=843810
BC00402=843810
BC00403=902188
BC00404=900128
BC00405=900128
BC00406=900128
BC00407=900128
BC00408=900128
BC00409=963634
BC00410=965489
BC00411=965489
BC00412=965489
BC00413=965489
BC00414=965489
BC00415=965489
BC00416=965489
BC00417=965489
BC00418=965489
BC00419=965489
BC00420=965489
BC00421=995027
BC00422=1000860
BC00423=1000860
BC00424=1000860
BC00425=1000860
BC00426=1000860
BC00427=965489
BC00428=981769
BC00429=981769
BC00430=981769
BC00431=979574
BC00432=931504
BC00433=769966
BC00434=769966
BC00435=716686
BC00436=679663
BC00437=721442
BC00438=721442
BC00439=721439
BC00440=781482
BC00441=781888
BC00442=781888
BC00443=781888
BC00444=781888
BC00445=768943
BC00446=718475
BC00447=718475
BC00448=718475
BC00449=778313
BC00450=778313
BC00451=717855
BC00452=792672
BC00453=792672
BC00454=948195
BC00455=948195
BC00456=957587
BC00457=959389
BC00458=967513
BC00459=969988
BC00460=976572
BC00461=976572
BC00462=957101
BC00463=956675
BC00464=968192
BC00465=950199
BC00466=792672
BC00467=792672
BC00468=792672
BC00469=887446
BC00470=956264
BC00471=956264
BC00472=969252
BC00473=969531
BC00474=979980
BC00475=973562
BC00476=990042
BC00477=986050
BC00478=987878
BC00479=987878
BC00480=956264
BC00481=956264
BC00482=887446
BC00483=792672
BC00484=792672
BC00485=700249
BC00486=546214
BC00487=546214
BC00488=546211
BC00489=546211
BC00490=406776
BC00491=406776
BC00492=352261
BC00493=346119
BC00494=406266
BC00495=406266
BC00496=491556
BC00497=546211
BC00498=546214
BC00499=546214
BC00500=507604
BC00501=410782
BC00502=429690
BC00503=375447
BC00504=350474
BC00505=350474
BC00506=408658
BC00507=408658
BC00508=507604
BC00509=546214
BC00510=546214
BC00511=516757
BC00512=591809
BC00513=591809
BC00514=591809
BC00515=591183
BC00516=650353
BC00517=650538
BC00518=650538
BC00519=584003
BC00520=515801
BC00521=520018
BC00522=520018
BC00523=590597
BC00524=593080
BC00525=593080
BC00526=593080
BC00527=652365
BC00528=652559
BC00529=594501
BC00530=537666
BC00531=433888
BC00532=546211
BC00533=830322
BC00534=830322
BC00535=830322
BC00536=890247
BC00537=890396
BC00538=798848
BC00539=798848
BC00540=798848
BC00541=798848
BC00542=832296
BC00543=845010
BC00544=845010
BC00545=904605
BC00546=904704
BC00547=818840
BC00548=818839
BC00549=818839
BC00550=526967
BC00551=334612
BC00552=334612
BC00553=334612
BC00554=350464
BC00555=350464
BC00556=359337
BC00557=359337
BC00558=359337
BC00559=359337
BC00560=359453
BC00561=359337
BC00562=359337
BC00563=359337
BC00564=359337
BC00565=359337
BC00566=358620
BC00567=350464
BC00568=334612
BC00569=334612
BC00570=334612
BC00571=334613
BC00572=501279
BC00573=501279
BC00574=334612
BC00575=334610
BC00576=349510
BC00577=365935
BC00578=365935
BC00579=365934
BC00580=348430
BC00581=348430
BC00582=348430
BC00583=365935
BC00584=349510
BC00585=334610
BC00586=334612
BC00587=334612
BC00588=512789
BC00589=516757
BC00590=526627
BC00591=466969
BC00592=466969
BC00593=466969
BC00594=524647
BC00595=525745
BC00596=525745
BC00597=525745
BC00598=525745
BC00599=473911
BC00600=473911
BC00601=473911
BC00602=532824
BC00603=533743
BC00604=525745
BC00605=525745
BC00606=525747
///POSTYPE BASE
///RECTAN
///RCONF 1,0,0,0,0,0,0,0,0,0,0,0,0,0,0,0,0,0,0,0,0,0,0,0
P00006=0.000,0.000,0.000,0.0000,0.0000,0.0000
///RCONF 0,0,0,0,0,0,0,0,0,0,0,0,0,0,0,0,0,0,0,0,0,0,0,0
P00057=0.000,0.000,2.000,0.0000,0.0000,0.0000
P00058=0.000,0.000,3.000,0.0000,0.0000,0.0000
///RCONF 1,0,0,0,0,0,0,0,0,0,0,0,0,0,0,0,0,0,0,0,0,0,0,0
P00099=0.011,-2.380,1.226,0.0000,0.0000,0.0000
P00100=-0.081,2.558,4.482,0.0000,0.0000,0.0000
P00101=0.030,-2.286,2.993,0.0000,0.0000,0.0000
P00102=-0.005,-1.108,1.644,0.0000,0.0000,0.0000
P00103=-0.094,-3.400,4.200,0.0000,0.0000,0.0000
P00104=0.043,-2.127,5.826,0.0000,0.0000,0.0000
P00105=-0.043,0.662,5.286,0.0000,0.0000,0.0000
P00106=-0.018,-2.519,0.237,0.0000,0.0000,0.0000
P00107=-0.008,-4.537,-4.500,0.0000,0.0000,0.0000
P00108=0.014,-3.040,2.637,0.0000,0.0000,0.0000
///RCONF 0,0,0,0,0,0,0,0,0,0,0,0,0,0,0,0,0,0,0,0,0,0,0,0
P00299=-1.404,-0.874,9.133,0.0000,0.0000,0.0000
///RCONF 1,0,0,0,0,0,0,0,0,0,0,0,0,0,0,0,0,0,0,0,0,0,0,0
P00300=-0.036,-1.505,2.318,0.0000,0.0000,0.0000
P00301=0.046,-2.112,7.779,0.0000,0.0000,0.0000
P00302=-0.180,-2.409,6.326,0.0000,0.0000,0.0000
///RCONF 0,0,0,0,0,0,0,0,0,0,0,0,0,0,0,0,0,0,0,0,0,0,0,0
P00303=-0.004,-1.437,-4.584,0.0000,0.0000,0.0000
P00304=0.028,-1.666,-4.234,0.0000,0.0000,0.0000
P00305=-0.003,-1.920,-3.501,0.0000,0.0000,0.0000
P00306=0.015,-2.252,-3.054,0.0000,0.0000,0.0000
P00307=0.019,-2.151,-5.077,0.0000,0.0000,0.0000
P00308=-0.003,-2.092,-4.888,0.0000,0.0000,0.0000
P00309=-0.040,-2.205,-4.992,0.0000,0.0000,0.0000
P00310=-0.006,-2.490,-5.925,0.0000,0.0000,0.0000
P00311=-0.007,-2.079,-5.307,0.0000,0.0000,0.0000
P00312=-0.032,2.202,-7.632,0.0000,0.0000,0.0000
///RCONF 1,0,0,0,0,0,0,0,0,0,0,0,0,0,0,0,0,0,0,0,0,0,0,0
P00349=0.060,0.167,-1.133,0.0000,0.0000,0.0000
///RCONF 0,0,0,0,0,0,0,0,0,0,0,0,0,0,0,0,0,0,0,0,0,0,0,0
P00350=11.519,-0.008,1.149,0.0000,0.0000,0.0000
P00351=13.563,-0.027,-0.653,0.0000,0.0000,0.0000
P00352=13.252,-0.027,-0.827,0.0000,0.0000,0.0000
P00353=10.971,-0.082,0.776,0.0000,0.0000,0.0000
P00354=-0.024,2.508,-1.824,0.0000,0.0000,0.0000
P00355=-0.001,2.528,-1.131,0.0000,0.0000,0.0000
P00356=-0.034,2.921,-0.262,0.0000,0.0000,0.0000
P00357=0.003,3.386,-0.091,0.0000,0.0000,0.0000
P00358=0.014,3.037,-0.020,0.0000,0.0000,0.0000
P00359=-0.005,2.731,0.912,0.0000,0.0000,0.0000
P00360=-0.011,3.412,0.438,0.0000,0.0000,0.0000
P00361=0.018,3.050,1.253,0.0000,0.0000,0.0000
P00362=0.014,2.784,0.148,0.0000,0.0000,0.0000
P00399=-2.449,0.031,8.825,0.0000,0.0000,0.0000
P00400=5.920,-3.503,-0.024,0.0000,0.0000,0.0000
P00401=3.430,-0.021,1.131,0.0000,0.0000,0.0000
P00402=-0.253,1.107,3.062,0.0000,0.0000,0.0000
P00403=-3.666,-0.015,5.328,0.0000,0.0000,0.0000
P00405=2.420,0.007,1.427,0.0000,0.0000,0.0000
P00406=3.513,-0.022,0.429,0.0000,0.0000,0.0000
P00415=-1.781,-1.303,3.250,0.0000,0.0000,0.0000
P00416=0.027,1.119,3.078,0.0000,0.0000,0.0000
//INST
///DATE 2024/10/29 13:39
///ATTR SC,RW
///GROUP1 RB1,BS1
NOP
CALL JOB:MOVE_INTO_TUNNEL
SFTOF
'------------------------
'------------------------
'SPOINA SRODEK DOL
'------------------------
'------------------------
MOVJ C00000 BC00000 VJ=10.00
MOVJ C00001 BC00001 VJ=30.00
'------------------------
'W38 P
'------------------------
'TEST
MOVL C00002 BC00002 V=166.7
MOVL C00003 BC00003 V=166.7 PL=0
REFP 3 C00004 BC00004
CALL JOB:SEARCH-R1
IMOV P0057 V=23.0
SET P0099 P0006
SFTON P0099
REFP 3 C00005 BC00005
CALL JOB:SEARCH-R1
SET P0099 P0006
SFTON P0099
MOVL C00006 BC00006 V=166.7 PL=0
'TEST
SFTOF
MOVL C00007 BC00007 V=333.3
MOVL C00008 BC00008 V=333.3
'------------------------
'W38 L
'------------------------
'TEST
MOVL C00009 BC00009 V=166.7 PL=0
REFP 3 C00010 BC00010
CALL JOB:SEARCH-R1
IMOV P0057 V=23.0
SET P0100 P0006
SFTON P0100
REFP 3 C00011 BC00011
CALL JOB:SEARCH-R1
SET P0100 P0006
SFTON P0100
MOVL C00012 BC00012 V=166.7 PL=0
'TEST
SFTOF
MOVJ C00013 BC00013 VJ=20.00
'------------------------
'W45 P
'------------------------
MOVL C00014 BC00014 V=166.7 PL=0
REFP 3 C00015 BC00015
CALL JOB:SEARCH-R1
IMOV P0057 V=23.0
SET P0101 P0006
SFTON P0101
REFP 3 C00016 BC00016
CALL JOB:SEARCH-R1
SET P0101 P0006
SFTON P0101
MOVL C00017 BC00017 V=166.7 PL=0
'TEST
SFTOF
MOVJ C00018 BC00018 VJ=20.00
'------------------------
'W45 L
'------------------------
MOVL C00019 BC00019 V=133.3 PL=0
REFP 3 C00020 BC00020
CALL JOB:SEARCH-R1
IMOV P0057 V=23.0
SET P0102 P0006
SFTON P0102
REFP 3 C00021 BC00021
CALL JOB:SEARCH-R1
SET P0102 P0006
SFTON P0102
MOVL C00022 BC00022 V=250.0 PL=0
'TEST
SFTOF
MOVJ C00023 BC00023 VJ=20.00
'------------------------
'W48 P
'------------------------
'TEST
MOVL C00024 BC00024 V=133.3 PL=0
REFP 3 C00025 BC00025
CALL JOB:SEARCH-R1
IMOV P0057 V=23.0
SET P0103 P0006
SFTON P0103
REFP 3 C00026 BC00026
CALL JOB:SEARCH-R1
SET P0103 P0006
SFTON P0103
MOVL C00027 BC00027 V=166.7 PL=0
'TEST
SFTOF
MOVJ C00028 BC00028 VJ=30.00
MOVJ C00029 BC00029 VJ=30.00
MOVJ C00030 BC00030 VJ=30.00
MOVJ C00031 BC00031 VJ=30.00
MOVJ C00032 BC00032 VJ=20.00
MOVL C00033 BC00033 V=250.0
'------------------------
'W48 L
'------------------------
SFTOF
MOVL C00034 BC00034 V=133.3 PL=0
REFP 3 C00035 BC00035
CALL JOB:SEARCH-R1
IMOV P0057 V=23.0
SET P0104 P0006
SFTON P0104
REFP 3 C00036 BC00036
CALL JOB:SEARCH-R1
SET P0104 P0006
SFTON P0104
MOVL C00037 BC00037 V=166.7 PL=0
SFTOF
MOVJ C00038 BC00038 VJ=20.00
'------------------------
'W36 P
'------------------------
MOVL C00039 BC00039 V=133.3 PL=0
REFP 3 C00040 BC00040
CALL JOB:SEARCH-R1
IMOV P0057 V=23.0
SET P0105 P0006
SFTON P0105
REFP 3 C00041 BC00041
CALL JOB:SEARCH-R1
SET P0105 P0006
SFTON P0105
MOVL C00042 BC00042 V=166.7 PL=0
'TEST
SFTOF
MOVJ C00043 BC00043 VJ=20.00
'------------------------
'W36 L
'------------------------
MOVL C00044 BC00044 V=166.7 PL=0
REFP 3 C00045 BC00045
CALL JOB:SEARCH-R1
IMOV P0057 V=23.0
SET P0106 P0006
SFTON P0106
REFP 3 C00046 BC00046
CALL JOB:SEARCH-R1
SET P0106 P0006
SFTON P0106
MOVL C00047 BC00047 V=166.7 PL=0
'TEST
MOVJ C00048 BC00048 VJ=20.00
SFTOF
'------------------------
'W44 P
'------------------------
'TEST
MOVL C00049 BC00049 V=133.3 PL=0
REFP 3 C00050 BC00050
CALL JOB:SEARCH-R1
IMOV P0057 V=23.0
SET P0107 P0006
SFTON P0107
REFP 3 C00051 BC00051
CALL JOB:SEARCH-R1
SET P0107 P0006
SFTON P0107
MOVL C00052 BC00052 V=250.0 PL=0
'TEST
SFTOF
MOVL C00053 BC00053 V=250.0
MOVJ C00054 BC00054 VJ=25.00
MOVJ C00055 BC00055 VJ=25.00
MOVJ C00056 BC00056 VJ=25.00
MOVJ C00057 BC00057 VJ=25.00
MOVJ C00058 BC00058 VJ=30.00
MOVJ C00059 BC00059 VJ=25.00
'------------------------
'W44 L
'------------------------
'TEST
MOVL C00060 BC00060 V=166.7 PL=0
REFP 3 C00061 BC00061
CALL JOB:SEARCH-R1
IMOV P0057 V=23.0
SET P0108 P0006
SFTON P0108
REFP 3 C00062 BC00062
CALL JOB:SEARCH-R1
SET P0108 P0006
SFTON P0108
MOVL C00063 BC00063 V=250.0 PL=0
'TEST
SFTOF
MOVL C00064 BC00064 V=250.0
MOVJ C00065 BC00065 VJ=25.00
IFTHENEXP OT#(1457)=ON ANDEXP OT#(1441)=OFF
	 CALL JOB:TWIN_FRONT_WELD_-90ST-2_5340
ENDIF
IFTHENEXP OT#(1457)=OFF ANDEXP OT#(1441)=ON
	 CALL JOB:FRONT_SEARCH_0ST-2_5340
ENDIF
COMM MOVJ C00066 BC00066 VJ=20.00
COMM MOVJ C00067 BC00067 VJ=20.00
COMM MOVJ C00068 BC00068 VJ=20.00
COMM 'DODANE
COMM 'SZUKANIE FRONT
COMM '------------------------
COMM '503
COMM '------------------------
COMM MOVL C00069 BC00069 V=333.3
COMM MOVL C00070 BC00070 V=166.7 PL=0
COMM REFP 3 C00071 BC00071
COMM CALL JOB:SEARCH-R1
COMM IMOV P0058 V=16.7
COMM SET P0350 P0006
COMM SFTON P0350
COMM REFP 3 C00072 BC00072
COMM CALL JOB:SEARCH-R1
COMM SET P0350 P0006
COMM SFTON P0350
COMM MOVL C00073 BC00073 V=66.7 PL=0
COMM SFTOF
COMM '------------------------
COMM '------------------------
COMM '502
COMM '------------------------
COMM MOVL C00074 BC00074 V=166.7
COMM MOVL C00075 BC00075 V=66.7 PL=0
COMM REFP 3 C00076 BC00076
COMM CALL JOB:SEARCH-R1
COMM IMOV P0058 V=16.7
COMM SET P0351 P0006
COMM SFTON P0351
COMM REFP 3 C00077 BC00077
COMM CALL JOB:SEARCH-R1
COMM SET P0351 P0006
COMM SFTON P0351
COMM MOVL C00078 BC00078 V=66.7 PL=0
COMM SFTOF
COMM '------------------------
COMM '------------------------
COMM '501
COMM '------------------------
COMM MOVL C00079 BC00079 V=166.7
COMM MOVL C00080 BC00080 V=66.7 PL=0
COMM REFP 3 C00081 BC00081
COMM CALL JOB:SEARCH-R1
COMM IMOV P0058 V=16.7
COMM SET P0352 P0006
COMM SFTON P0352
COMM REFP 3 C00082 BC00082
COMM CALL JOB:SEARCH-R1
COMM SET P0352 P0006
COMM SFTON P0352
COMM MOVL C00083 BC00083 V=66.7 PL=0
COMM SFTOF
COMM '------------------------
COMM '------------------------
COMM '500
COMM '------------------------
COMM MOVL C00084 BC00084 V=166.7
COMM MOVL C00085 BC00085 V=66.7 PL=0
COMM REFP 3 C00086 BC00086
COMM CALL JOB:SEARCH-R1
COMM IMOV P0058 V=16.7
COMM SET P0353 P0006
COMM SFTON P0353
COMM REFP 3 C00087 BC00087
COMM CALL JOB:SEARCH-R1
COMM SET P0353 P0006
COMM SFTON P0353
COMM MOVL C00088 BC00088 V=66.7 PL=0
COMM SFTOF
COMM '------------------------
COMM MOVL C00089 BC00089 V=333.3
COMM MOVL C00090 BC00090 V=333.3
COMM MOVJ C00091 BC00091 VJ=10.00
COMM 'DODANE
COMM MOVJ C00092 BC00092 VJ=10.00
COMM '------------------------
COMM 'SFT402
COMM '------------------------
COMM SFTOF
COMM MOVL C00093 BC00093 V=150.0
COMM MOVL C00094 BC00094 V=66.7 PL=0
COMM REFP 3 C00095 BC00095
COMM CALL JOB:SEARCH-R1
COMM SET P0402 P0006
COMM SFTON P0402
COMM MOVL C00096 BC00096 V=150.0
COMM MOVL C00097 BC00097 V=66.7 PL=0
COMM REFP 3 C00098 BC00098
COMM CALL JOB:SEARCH-R1
COMM SET P0402 P0006
COMM SFTON P0402
COMM MOVL C00099 BC00099 V=133.3
COMM MOVL C00100 BC00100 V=150.0
COMM MOVL C00101 BC00101 V=150.0
COMM MOVL C00102 BC00102 V=66.7 PL=0
COMM REFP 3 C00103 BC00103
COMM CALL JOB:SEARCH-R1
COMM SET P0402 P0006
COMM SFTOF
COMM MOVL C00104 BC00104 V=150.0
COMM '------------------------
COMM 'SFT403
COMM '------------------------
COMM 'START
COMM SFTOF
COMM MOVL C00105 BC00105 V=250.0
COMM MOVL C00106 BC00106 V=133.3 PL=0
COMM REFP 3 C00107 BC00107
COMM CALL JOB:SEARCH-R1
COMM SET P0416 P0006
COMM SFTON P0416
COMM MOVL C00108 BC00108 V=133.3
COMM REFP 3 C00109 BC00109
COMM CALL JOB:SEARCH-R1
COMM SET P0402 P0006
COMM SFTOF
COMM MOVL C00110 BC00110 V=150.0
COMM '------------------------
COMM '------------------------
COMM SFTOF
COMM MOVL C00111 BC00111 V=250.0
COMM MOVL C00112 BC00112 V=133.3 PL=0
COMM REFP 3 C00113 BC00113
COMM CALL JOB:SEARCH-R1
COMM SET P0403 P0006
COMM SFTON P0403
COMM MOVL C00114 BC00114 V=66.7 PL=0
COMM REFP 3 C00115 BC00115
COMM CALL JOB:SEARCH-R1
COMM SET P0403 P0006
COMM SFTOF
COMM MOVL C00116 BC00116 V=150.0
COMM MOVJ C00117 BC00117 VJ=20.00
COMM MOVJ C00118 BC00118 VJ=20.00
COMM '------------------------
COMM 'SFT401
COMM '------------------------
COMM SFTOF
COMM MOVL C00119 BC00119 V=150.0
COMM MOVL C00120 BC00120 V=66.7 PL=0
COMM REFP 3 C00121 BC00121
COMM CALL JOB:SEARCH-R1
COMM SET P0401 P0006
COMM SFTON P0401
COMM MOVL C00122 BC00122 V=66.7 PL=0
COMM REFP 3 C00123 BC00123
COMM CALL JOB:SEARCH-R1
COMM SET P0401 P0006
COMM SFTOF
COMM MOVL C00124 BC00124 V=150.0
COMM 'SFT400
COMM '------------------------
COMM SFTOF
COMM MOVL C00125 BC00125 V=333.3
COMM MOVL C00126 BC00126 V=66.7 PL=0
COMM REFP 3 C00127 BC00127
COMM CALL JOB:SEARCH-R1
COMM SET P0405 P0006
COMM SFTON P0405
COMM MOVL C00128 BC00128 V=66.7 PL=0
COMM REFP 3 C00129 BC00129
COMM CALL JOB:SEARCH-R1
COMM SET P0405 P0006
COMM SFTOF
COMM MOVL C00130 BC00130 V=150.0
COMM 'SFT400
COMM '------------------------
COMM SFTOF
COMM MOVL C00131 BC00131 V=333.3
COMM MOVL C00132 BC00132 V=133.3 PL=0
COMM REFP 3 C00133 BC00133
COMM CALL JOB:SEARCH-R1
COMM SET P0406 P0006
COMM SFTON P0406
COMM MOVL C00134 BC00134 V=66.7 PL=0
COMM REFP 3 C00135 BC00135
COMM CALL JOB:SEARCH-R1
COMM SET P0406 P0006
COMM SFTOF
COMM MOVL C00136 BC00136 V=150.0
COMM 'SFT400
COMM '------------------------
COMM SFTOF
COMM MOVL C00137 BC00137 V=150.0
COMM MOVL C00138 BC00138 V=66.7 PL=0
COMM REFP 3 C00139 BC00139
COMM CALL JOB:SEARCH-R1
COMM SET P0400 P0006
COMM SFTON P0400
COMM MOVL C00140 BC00140 V=150.0
COMM MOVL C00141 BC00141 V=66.7 PL=0
COMM REFP 3 C00142 BC00142
COMM CALL JOB:SEARCH-R1
COMM SET P0400 P0006
COMM SFTON P0400
COMM MOVL C00143 BC00143 V=150.0
COMM MOVL C00144 BC00144 V=150.0
COMM MOVL C00145 BC00145 V=66.7 PL=0
COMM REFP 3 C00146 BC00146
COMM CALL JOB:SEARCH-R1
COMM SET P0400 P0006
COMM SFTOF
COMM MOVL C00147 BC00147 V=83.3
COMM MOVL C00148 BC00148 V=250.0
COMM MOVL C00149 BC00149 V=333.3
COMM MOVL C00150 BC00150 V=66.7 PL=0
COMM REFP 3 C00151 BC00151
COMM CALL JOB:SEARCH-R1
COMM SET P0415 P0006
COMM SFTON P0415
COMM MOVL C00152 BC00152 V=133.3
COMM REFP 3 C00153 BC00153
COMM CALL JOB:SEARCH-R1
COMM SET P0415 P0006
COMM SFTOF
COMM MOVL C00154 BC00154 V=150.0
COMM '------------------------
COMM 'SFT403
COMM '------------------------
COMM 'START
COMM SFTOF
COMM MOVJ C00155 BC00155 VJ=10.00
COMM '------------------------
COMM 'SFT399
COMM '------------------------
COMM 'START
COMM SFTOF
COMM MOVL C00156 BC00156 V=150.0
COMM MOVL C00157 BC00157 V=66.7 PL=0
COMM REFP 3 C00158 BC00158
COMM CALL JOB:SEARCH-R1
COMM SET P0399 P0006
COMM SFTON P0399
COMM MOVL C00159 BC00159 V=66.7 PL=0
COMM REFP 3 C00160 BC00160
COMM CALL JOB:SEARCH-R1
COMM SET P0399 P0006
COMM SFTOF
COMM MOVL C00161 BC00161 V=150.0
COMM MOVJ C00162 BC00162 VJ=20.00
COMM MOVJ C00163 BC00163 VJ=30.00
MOVJ C00164 BC00164 VJ=30.00
MOVJ C00165 BC00165 VJ=30.00
MOVJ C00166 BC00166 VJ=40.00
'WELD
'WELD
MOVJ C00167 BC00167 VJ=20.00
'**********************
'W36
'**********************
MOVL C00168 BC00168 V=500.0
SFTON P0105
MOVL C00169 BC00169 V=166.7 PL=0
SFTOF
MACRO1 MJ#(0) ARGF24
ARCON
SFTON P0106
MOVL C00170 BC00170 V=11.7
ARCOF
SFTOF
MOVJ C00171 BC00171 VJ=15.00
MOVJ C00172 BC00172 VJ=10.00
MOVJ C00173 BC00173 VJ=10.00
MOVJ C00174 BC00174 VJ=10.00
MOVJ C00175 BC00175 VJ=30.00
MOVJ C00176 BC00176 VJ=20.00
MOVJ C00177 BC00177 VJ=10.00
MOVJ C00178 BC00178 VJ=15.00
'**********************
'W38
'**********************
MOVL C00179 BC00179 V=500.0
SFTON P0100
MOVL C00180 BC00180 V=166.7 PL=0
SFTOF
ARCON
SFTON P0099
MOVL C00181 BC00181 V=11.3
ARCOF
SFTOF
'DODANE
MOVL C00182 BC00182 V=500.0
MOVJ C00183 BC00183 VJ=10.00
MOVJ C00184 BC00184 VJ=10.00
MOVJ C00185 BC00185 VJ=10.00
MOVJ C00186 BC00186 VJ=10.00
MOVJ C00187 BC00187 VJ=25.00
MOVJ C00188 BC00188 VJ=30.00
MOVJ C00189 BC00189 VJ=30.00
MOVJ C00190 BC00190 VJ=30.00
MOVL C00191 BC00191 V=500.0
SFTON P0107
MOVL C00192 BC00192 V=166.7 PL=0
SFTOF
MACRO1 MJ#(0) ARGF24
ARCON
SFTON P0108
MOVL C00193 BC00193 V=10.8
MOVL C00194 BC00194 V=10.8
ARCOF
SFTOF
MOVL C00195 BC00195 V=500.0
MOVL C00196 BC00196 V=500.0
MOVJ C00197 BC00197 VJ=10.00
MOVJ C00198 BC00198 VJ=10.00
MOVJ C00199 BC00199 VJ=20.00
'**********************
'DODATEK
'**********************
MOVJ C00200 BC00200 VJ=10.00
MOVJ C00201 BC00201 VJ=10.00
MOVJ C00202 BC00202 VJ=20.00
MOVJ C00203 BC00203 VJ=20.00
MOVJ C00204 BC00204 VJ=20.00
MOVL C00205 BC00205 V=333.3
MOVL C00206 BC00206 V=166.7
MACRO1 MJ#(0) ARGF24
SFTON P0108
MOVL C00207 BC00207 V=166.7 PL=0
SFTOF
ARCON
SFTON P0108
MOVL C00208 BC00208 V=10.8
ARCOF
SFTOF
MOVL C00209 BC00209 V=500.0
MOVJ C00210 BC00210 VJ=20.00
MOVJ C00211 BC00211 VJ=30.00
'**********************
'W45
'**********************
MOVJ C00212 BC00212 VJ=30.00
MOVJ C00213 BC00213 VJ=20.00
MOVJ C00214 BC00214 VJ=10.00
MACRO1 MJ#(0) ARGF24
MOVL C00215 BC00215 V=500.0
SFTON P0102
MOVL C00216 BC00216 V=166.7 PL=0
SFTOF
ARCON
SFTON P0101
MOVL C00217 BC00217 V=10.8
ARCOF
SFTOF
MOVL C00218 BC00218 V=500.0
MOVJ C00219 BC00219 VJ=10.00
MOVJ C00220 BC00220 VJ=10.00
'**********************
'W48
'**********************
MOVJ C00221 BC00221 VJ=15.00
MOVJ C00222 BC00222 VJ=15.00
MOVJ C00223 BC00223 VJ=15.00
SFTON P0103
MOVL C00224 BC00224 V=166.7 PL=0
SFTOF
ARCON
SFTON P0104
MOVL C00225 BC00225 V=10.8
ARCOF
SFTOF
MOVL C00226 BC00226 V=500.0
MOVJ C00227 BC00227 VJ=15.00
MOVJ C00228 BC00228 VJ=20.00
MOVJ C00229 BC00229 VJ=40.00
IFTHENEXP OT#(1457)=ON ANDEXP OT#(1441)=OFF
	 CALL JOB:TWIN_FRONT_WELD_0ST-2_5340
ENDIF
IFTHENEXP OT#(1457)=OFF ANDEXP OT#(1441)=ON
	 CALL JOB:FRONT_WELD_0ST-2_5340
ENDIF
MOVL C00230 BC00230 V=333.3
CALL JOB:MOVE_OUT_OF_TUNNEL
CALL JOB:CLEAN-R1
CALL JOB:MOVE_INTO_TUNNEL
MOVJ C00231 BC00231 VJ=30.00 PL=0
'------------------------
'------------------------
'PRAWA STRONA PROFIL GORA
'------------------------
'------------------------
MOVJ C00232 BC00232 VJ=20.00
'------------------------
'W51A L
'------------------------
SFTOF
MOVJ C00233 BC00233 VJ=10.00
MOVL C00234 BC00234 V=66.7 PL=0
REFP 3 C00235 BC00235
CALL JOB:SEARCH-R1
SET P0299 P0006
SFTON P0299
MOVL C00236 BC00236 V=66.7 PL=0
REFP 3 C00237 BC00237
CALL JOB:SEARCH-R1
SET P0299 P0006
SFTON P0299
MOVL C00238 BC00238 V=83.3
MOVL C00239 BC00239 V=166.7 PL=0
REFP 3 C00240 BC00240
CALL JOB:SEARCH-R1
SET P0299 P0006
SFTON P0299
MOVL C00241 BC00241 V=133.3 PL=0
SFTOF
'------------------------
'W51A P
'------------------------
SFTOF
MOVL C00242 BC00242 V=250.0
MOVL C00243 BC00243 V=66.7 PL=0
REFP 3 C00244 BC00244
CALL JOB:SEARCH-R1
SET P0300 P0006
SFTON P0300
MOVL C00245 BC00245 V=66.7 PL=0
REFP 3 C00246 BC00246
CALL JOB:SEARCH-R1
SET P0300 P0006
SFTON P0300
MOVL C00247 BC00247 V=66.7 PL=0
SFTOF
'------------------------
'W54A L
'------------------------
SFTOF
MOVJ C00248 BC00248 VJ=30.00
MOVL C00249 BC00249 V=133.3 PL=0
REFP 3 C00250 BC00250
CALL JOB:SEARCH-R1
SET P0301 P0006
SFTON P0301
MOVL C00251 BC00251 V=66.7 PL=0
REFP 3 C00252 BC00252
CALL JOB:SEARCH-R1
SET P0301 P0006
SFTON P0301
MOVL C00253 BC00253 V=66.7 PL=0
SFTOF
'------------------------
'W54A P
'------------------------
SFTOF
MOVJ C00254 BC00254 VJ=30.00
MOVL C00255 BC00255 V=133.3 PL=0
REFP 3 C00256 BC00256
CALL JOB:SEARCH-R1
SET P0302 P0006
SFTON P0302
MOVL C00257 BC00257 V=66.7 PL=0
REFP 3 C00258 BC00258
CALL JOB:SEARCH-R1
SET P0302 P0006
SFTON P0302
MOVL C00259 BC00259 V=66.7 PL=0
SFTOF
'------------------------
'W50A L
'------------------------
SFTOF
MOVJ C00260 BC00260 VJ=30.00
MOVL C00261 BC00261 V=133.3 PL=0
REFP 3 C00262 BC00262
CALL JOB:SEARCH-R1
SET P0303 P0006
SFTON P0303
MOVL C00263 BC00263 V=66.7 PL=0
REFP 3 C00264 BC00264
CALL JOB:SEARCH-R1
SET P0303 P0006
SFTON P0303
MOVL C00265 BC00265 V=66.7 PL=0
SFTOF
'------------------------
'W50A P
'------------------------
SFTOF
MOVJ C00266 BC00266 VJ=30.00
MOVL C00267 BC00267 V=133.3 PL=0
REFP 3 C00268 BC00268
CALL JOB:SEARCH-R1
SET P0304 P0006
SFTON P0304
MOVL C00269 BC00269 V=66.7 PL=0
REFP 3 C00270 BC00270
CALL JOB:SEARCH-R1
SET P0304 P0006
SFTON P0304
MOVL C00271 BC00271 V=66.7 PL=0
SFTOF
'------------------------
'W53A L
'------------------------
SFTOF
MOVJ C00272 BC00272 VJ=30.00
MOVL C00273 BC00273 V=133.3 PL=0
REFP 3 C00274 BC00274
CALL JOB:SEARCH-R1
SET P0305 P0006
SFTON P0305
MOVL C00275 BC00275 V=66.7 PL=0
REFP 3 C00276 BC00276
CALL JOB:SEARCH-R1
SET P0305 P0006
SFTON P0305
MOVL C00277 BC00277 V=66.7 PL=0
SFTOF
'------------------------
'W53A P
'------------------------
SFTOF
MOVJ C00278 BC00278 VJ=30.00
MOVL C00279 BC00279 V=200.0
MOVL C00280 BC00280 V=66.7 PL=0
REFP 3 C00281 BC00281
CALL JOB:SEARCH-R1
SET P0306 P0006
SFTON P0306
MOVL C00282 BC00282 V=66.7 PL=0
REFP 3 C00283 BC00283
CALL JOB:SEARCH-R1
SET P0306 P0006
SFTON P0306
MOVL C00284 BC00284 V=66.7 PL=0
SFTOF
'------------------------
'W56A L
'------------------------
SFTOF
MOVJ C00285 BC00285 VJ=30.00
MOVL C00286 BC00286 V=133.3 PL=0
REFP 3 C00287 BC00287
CALL JOB:SEARCH-R1
SET P0307 P0006
SFTON P0307
MOVL C00288 BC00288 V=66.7 PL=0
REFP 3 C00289 BC00289
CALL JOB:SEARCH-R1
SET P0307 P0006
SFTON P0307
MOVL C00290 BC00290 V=66.7 PL=0
SFTOF
'------------------------
'W56A P
'------------------------
SFTOF
MOVJ C00291 BC00291 VJ=30.00
MOVL C00292 BC00292 V=133.3 PL=0
REFP 3 C00293 BC00293
CALL JOB:SEARCH-R1
SET P0308 P0006
SFTON P0308
MOVL C00294 BC00294 V=66.7 PL=0
REFP 3 C00295 BC00295
CALL JOB:SEARCH-R1
SET P0308 P0006
SFTON P0308
MOVL C00296 BC00296 V=66.7 PL=0
SFTOF
'------------------------
'W52A L
'------------------------
SFTOF
MOVJ C00297 BC00297 VJ=30.00
MOVL C00298 BC00298 V=250.0
MOVL C00299 BC00299 V=66.7 PL=0
REFP 3 C00300 BC00300
CALL JOB:SEARCH-R1
SET P0309 P0006
SFTON P0309
MOVL C00301 BC00301 V=66.7 PL=0
REFP 3 C00302 BC00302
CALL JOB:SEARCH-R1
SET P0309 P0006
SFTON P0309
MOVL C00303 BC00303 V=66.7 PL=0
SFTOF
'------------------------
'W52A P
'------------------------
SFTOF
MOVJ C00304 BC00304 VJ=5.00
MOVJ C00305 BC00305 VJ=20.00
MOVL C00306 BC00306 V=116.7 PL=0
REFP 3 C00307 BC00307
CALL JOB:SEARCH-R1
SET P0310 P0006
SFTON P0310
MOVL C00308 BC00308 V=66.7 PL=0
REFP 3 C00309 BC00309
CALL JOB:SEARCH-R1
SET P0310 P0006
SFTON P0310
MOVL C00310 BC00310 V=66.7 PL=0
SFTOF
'------------------------
'W55A L
'------------------------
SFTOF
MOVL C00311 BC00311 V=250.0
MOVJ C00312 BC00312 VJ=10.00
MOVL C00313 BC00313 V=66.7 PL=0
REFP 3 C00314 BC00314
CALL JOB:SEARCH-R1
SET P0311 P0006
SFTON P0311
MOVL C00315 BC00315 V=66.7 PL=0
REFP 3 C00316 BC00316
CALL JOB:SEARCH-R1
SET P0311 P0006
SFTON P0311
MOVL C00317 BC00317 V=66.7 PL=0
SFTOF
'------------------------
'W55A P
'------------------------
SFTOF
MOVL C00318 BC00318 V=250.0
MOVL C00319 BC00319 V=166.7
MOVL C00320 BC00320 V=66.7 PL=0
REFP 3 C00321 BC00321
CALL JOB:SEARCH-R1
SET P0312 P0006
SFTON P0312
MOVL C00322 BC00322 V=66.7 PL=0
REFP 3 C00323 BC00323
CALL JOB:SEARCH-R1
SET P0312 P0006
SFTON P0312
MOVL C00324 BC00324 V=66.7 PL=0
MOVL C00325 BC00325 V=166.7
SFTOF
MOVL C00326 BC00326 V=250.0
MOVJ C00327 BC00327 VJ=20.00
MOVJ C00328 BC00328 VJ=20.00
MOVJ C00329 BC00329 VJ=20.00
MOVJ C00330 BC00330 VJ=20.00
MOVJ C00331 BC00331 VJ=20.00
MOVJ C00332 BC00332 VJ=20.00
'------------------------
'------------------------
'LEWA STRONA PROFIL GORA
'------------------------
'------------------------
MOVJ C00333 BC00333 VJ=10.00
'------------------------
'W55B L
'------------------------
SFTOF
MOVJ C00334 BC00334 VJ=10.00
MOVL C00335 BC00335 V=66.7 PL=0
REFP 3 C00336 BC00336
CALL JOB:SEARCH-R1
SET P0349 P0006
SFTON P0349
MOVL C00337 BC00337 V=66.7 PL=0
REFP 3 C00338 BC00338
CALL JOB:SEARCH-R1
SET P0349 P0006
SFTON P0349
MOVL C00339 BC00339 V=66.7 PL=0
SFTOF
MOVJ C00340 BC00340 VJ=10.00
MOVJ C00341 BC00341 VJ=10.00
'------------------------
'W55B P
'------------------------
SFTOF
MOVL C00342 BC00342 V=66.7 PL=0
REFP 3 C00343 BC00343
CALL JOB:SEARCH-R1
SET P0350 P0006
SFTON P0350
MOVL C00344 BC00344 V=66.7 PL=0
REFP 3 C00345 BC00345
CALL JOB:SEARCH-R1
SET P0350 P0006
SFTON P0350
MOVL C00346 BC00346 V=66.7 PL=0
SFTOF
'------------------------
'W52B L
'------------------------
SFTOF
MOVJ C00347 BC00347 VJ=20.00
MOVJ C00348 BC00348 VJ=20.00
MOVL C00349 BC00349 V=150.0
MOVL C00350 BC00350 V=66.7 PL=0
REFP 3 C00351 BC00351
CALL JOB:SEARCH-R1
SET P0351 P0006
SFTON P0351
MOVL C00352 BC00352 V=66.7 PL=0
REFP 3 C00353 BC00353
CALL JOB:SEARCH-R1
SET P0351 P0006
SFTON P0351
MOVL C00354 BC00354 V=66.7 PL=0
SFTOF
'------------------------
'W52B P
'------------------------
SFTOF
MOVJ C00355 BC00355 VJ=30.00
MOVL C00356 BC00356 V=116.7 PL=0
REFP 3 C00357 BC00357
CALL JOB:SEARCH-R1
SET P0352 P0006
SFTON P0352
MOVL C00358 BC00358 V=66.7 PL=0
REFP 3 C00359 BC00359
CALL JOB:SEARCH-R1
SET P0352 P0006
SFTON P0352
MOVL C00360 BC00360 V=66.7 PL=0
SFTOF
'------------------------
'W56B L
'------------------------
SFTOF
MOVJ C00361 BC00361 VJ=30.00
MOVL C00362 BC00362 V=116.7 PL=0
REFP 3 C00363 BC00363
CALL JOB:SEARCH-R1
SET P0353 P0006
SFTON P0353
MOVL C00364 BC00364 V=66.7 PL=0
REFP 3 C00365 BC00365
CALL JOB:SEARCH-R1
SET P0353 P0006
SFTON P0353
MOVL C00366 BC00366 V=66.7 PL=0
SFTOF
'------------------------
'W56B P
'------------------------
SFTOF
MOVJ C00367 BC00367 VJ=30.00
MOVL C00368 BC00368 V=116.7 PL=0
REFP 3 C00369 BC00369
CALL JOB:SEARCH-R1
SET P0354 P0006
SFTON P0354
MOVL C00370 BC00370 V=66.7 PL=0
REFP 3 C00371 BC00371
CALL JOB:SEARCH-R1
SET P0354 P0006
SFTON P0354
MOVL C00372 BC00372 V=66.7 PL=0
SFTOF
'------------------------
'W53B L
'------------------------
SFTOF
MOVJ C00373 BC00373 VJ=30.00
MOVL C00374 BC00374 V=116.7 PL=0
REFP 3 C00375 BC00375
CALL JOB:SEARCH-R1
SET P0355 P0006
SFTON P0355
MOVL C00376 BC00376 V=66.7 PL=0
REFP 3 C00377 BC00377
CALL JOB:SEARCH-R1
SET P0355 P0006
SFTON P0355
MOVL C00378 BC00378 V=66.7 PL=0
SFTOF
'------------------------
'W53B P
'------------------------
SFTOF
MOVJ C00379 BC00379 VJ=30.00
MOVL C00380 BC00380 V=116.7 PL=0
REFP 3 C00381 BC00381
CALL JOB:SEARCH-R1
SET P0356 P0006
SFTON P0356
MOVL C00382 BC00382 V=66.7 PL=0
REFP 3 C00383 BC00383
CALL JOB:SEARCH-R1
SET P0356 P0006
SFTON P0356
MOVL C00384 BC00384 V=66.7 PL=0
SFTOF
'------------------------
'W50B L
'------------------------
SFTOF
MOVJ C00385 BC00385 VJ=30.00
MOVL C00386 BC00386 V=116.7 PL=0
REFP 3 C00387 BC00387
CALL JOB:SEARCH-R1
SET P0357 P0006
SFTON P0357
MOVL C00388 BC00388 V=66.7 PL=0
REFP 3 C00389 BC00389
CALL JOB:SEARCH-R1
SET P0357 P0006
SFTON P0357
MOVL C00390 BC00390 V=66.7 PL=0
SFTOF
'------------------------
'W50B P
'------------------------
SFTOF
MOVJ C00391 BC00391 VJ=30.00
MOVL C00392 BC00392 V=116.7 PL=0
REFP 3 C00393 BC00393
CALL JOB:SEARCH-R1
SET P0358 P0006
SFTON P0358
MOVL C00394 BC00394 V=66.7 PL=0
REFP 3 C00395 BC00395
CALL JOB:SEARCH-R1
SET P0358 P0006
SFTON P0358
MOVL C00396 BC00396 V=66.7 PL=0
SFTOF
'------------------------
'W54B L
'------------------------
SFTOF
MOVJ C00397 BC00397 VJ=30.00
MOVL C00398 BC00398 V=116.7 PL=0
REFP 3 C00399 BC00399
CALL JOB:SEARCH-R1
SET P0359 P0006
SFTON P0359
MOVL C00400 BC00400 V=66.7 PL=0
REFP 3 C00401 BC00401
CALL JOB:SEARCH-R1
SET P0359 P0006
SFTON P0359
MOVL C00402 BC00402 V=66.7 PL=0
SFTOF
'------------------------
'W54B P
'------------------------
SFTOF
MOVJ C00403 BC00403 VJ=30.00
MOVL C00404 BC00404 V=116.7 PL=0
REFP 3 C00405 BC00405
CALL JOB:SEARCH-R1
SET P0360 P0006
SFTON P0360
MOVL C00406 BC00406 V=66.7 PL=0
REFP 3 C00407 BC00407
CALL JOB:SEARCH-R1
SET P0360 P0006
SFTON P0360
MOVL C00408 BC00408 V=66.7 PL=0
SFTOF
'------------------------
'W51B L
'------------------------
SFTOF
MOVJ C00409 BC00409 VJ=30.00
MOVL C00410 BC00410 V=133.3 PL=0
REFP 3 C00411 BC00411
CALL JOB:SEARCH-R1
SET P0361 P0006
SFTON P0361
MOVL C00412 BC00412 V=66.7 PL=0
REFP 3 C00413 BC00413
CALL JOB:SEARCH-R1
SET P0361 P0006
SFTON P0361
MOVL C00414 BC00414 V=66.7 PL=0
SFTOF
'------------------------
'W51B P
'------------------------
SFTOF
MOVL C00415 BC00415 V=150.0
MOVL C00416 BC00416 V=66.7 PL=0
REFP 3 C00417 BC00417
CALL JOB:SEARCH-R1
SET P0361 P0006
SFTON P0361
MOVL C00418 BC00418 V=66.7 PL=0
REFP 3 C00419 BC00419
CALL JOB:SEARCH-R1
SET P0361 P0006
SFTON P0361
MOVL C00420 BC00420 V=166.7
SFTOF
MOVL C00421 BC00421 V=166.7
MOVL C00422 BC00422 V=66.7 PL=0
REFP 3 C00423 BC00423
CALL JOB:SEARCH-R1
SET P0362 P0006
SFTON P0362
MOVL C00424 BC00424 V=66.7 PL=0
REFP 3 C00425 BC00425
CALL JOB:SEARCH-R1
SET P0362 P0006
SFTON P0362
MOVL C00426 BC00426 V=83.3
MOVL C00427 BC00427 V=133.3 PL=0
MOVL C00428 BC00428 V=166.7
REFP 3 C00429 BC00429
CALL JOB:SEARCH-R1
SET P0362 P0006
SFTON P0362
SFTOF
MOVL C00430 BC00430 V=83.3
MOVL C00431 BC00431 V=250.0
MOVJ C00432 BC00432 VJ=20.00
MOVJ C00433 BC00433 VJ=30.00
MOVJ C00434 BC00434 VJ=10.00
MOVJ C00435 BC00435 VJ=40.00
'**********************
'**********************
'POCZATEK SPAWANIA BOKI
'**********************
'**********************
MOVJ C00436 BC00436 VJ=30.00
MOVJ C00437 BC00437 VJ=20.00
'**********************
'W50A
'**********************
MOVL C00438 BC00438 V=250.0
SFTON P0304
MOVL C00439 BC00439 V=83.3 PL=0
SFTOF
MACRO1 MJ#(0) ARGF10
ARCON
SFTON P0303
MOVL C00440 BC00440 V=10.8
ARCOF
SFTOF
MOVL C00441 BC00441 V=250.0
'W13B
MOVJ C00442 BC00442 VJ=20.00
MOVJ C00443 BC00443 VJ=40.00
MOVJ C00444 BC00444 VJ=20.00
MOVJ C00445 BC00445 VJ=20.00
MOVJ C00446 BC00446 VJ=20.00
'**********************
'W50B
'**********************
MOVL C00447 BC00447 V=250.0
SFTON P0357
MOVL C00448 BC00448 V=166.7 PL=0
SFTOF
MACRO1 MJ#(0) ARGF10
ARCON
SFTON P0358
MOVL C00449 BC00449 V=10.8
ARCOF
SFTOF
MOVL C00450 BC00450 V=250.0
MOVJ C00451 BC00451 VJ=20.00
MOVJ C00452 BC00452 VJ=20.00
MOVJ C00453 BC00453 VJ=20.00
MOVJ C00454 BC00454 VJ=20.00
'**********************
'W51A
'**********************
MOVL C00455 BC00455 V=416.7
MOVL C00456 BC00456 V=416.7
SFTON P0300
MOVL C00457 BC00457 V=166.7 PL=0
SFTOF
MACRO1 MJ#(0) ARGF10
ARCON
SFTON P0299
MOVL C00458 BC00458 V=10.8
MOVL C00459 BC00459 V=10.8
MOVL C00460 BC00460 V=10.8
MOVL C00461 BC00461 V=10.8
ARCOF
MOVL C00462 BC00462 V=166.7
MOVL C00463 BC00463 V=133.3 PL=0
ARCON
MOVL C00464 BC00464 V=8.3
ARCOF
SFTOF
MOVL C00465 BC00465 V=200.0
MOVJ C00466 BC00466 VJ=30.00
MOVJ C00467 BC00467 VJ=30.00
MOVJ C00468 BC00468 VJ=30.00
MOVJ C00469 BC00469 VJ=30.00
MOVJ C00470 BC00470 VJ=30.00
'**********************
'W51B
'**********************
MOVL C00471 BC00471 V=416.7
MOVL C00472 BC00472 V=416.7
SFTON P0361
MOVL C00473 BC00473 V=166.7 PL=0
SFTOF
MACRO1 MJ#(0) ARGF10
ARCON
SFTON P0362
MOVL C00474 BC00474 V=10.8
SFTON P0362
MOVL C00475 BC00475 V=10.8
MOVL C00476 BC00476 V=10.8
ARCOF
MOVL C00477 BC00477 V=166.7
MACRO1 MJ#(0) ARGF9
MOVL C00478 BC00478 V=166.7 PL=0
ARCON
MOVL C00479 BC00479 V=8.3
ARCOF
SFTOF
MOVL C00480 BC00480 V=166.7
MOVL C00481 BC00481 V=250.0
MOVJ C00482 BC00482 VJ=30.00
MOVJ C00483 BC00483 VJ=30.00
MOVJ C00484 BC00484 VJ=30.00
MOVJ C00485 BC00485 VJ=40.00
MOVJ C00486 BC00486 VJ=40.00
MOVJ C00487 BC00487 VJ=20.00
MOVJ C00488 BC00488 VJ=20.00
MOVJ C00489 BC00489 VJ=20.00
MOVJ C00490 BC00490 VJ=20.00
MOVJ C00491 BC00491 VJ=20.00
'**********************
'W52A
'**********************
SFTON P0310
MOVL C00492 BC00492 V=250.0
MOVL C00493 BC00493 V=83.3 PL=0
SFTOF
MACRO1 MJ#(0) ARGF10
ARCON
SFTON P0309
MOVL C00494 BC00494 V=10.8
ARCOF
SFTOF
MOVL C00495 BC00495 V=333.3
MOVJ C00496 BC00496 VJ=30.00
MOVJ C00497 BC00497 VJ=30.00
MOVJ C00498 BC00498 VJ=30.00
MOVJ C00499 BC00499 VJ=30.00
MOVJ C00500 BC00500 VJ=30.00
MOVJ C00501 BC00501 VJ=20.00
MOVJ C00502 BC00502 VJ=20.00
MOVJ C00503 BC00503 VJ=20.00
'**********************
'52B
'**********************
MOVL C00504 BC00504 V=250.0
SFTON P0351
MOVL C00505 BC00505 V=83.3 PL=0
SFTOF
MACRO1 MJ#(0) ARGF10
ARCON
SFTON P0352
MOVL C00506 BC00506 V=10.8
ARCOF
MOVL C00507 BC00507 V=333.3
SFTOF
MOVJ C00508 BC00508 VJ=20.00
MOVJ C00509 BC00509 VJ=30.00
MOVJ C00510 BC00510 VJ=30.00
'**********************
'W53A
'**********************
MOVJ C00511 BC00511 VJ=30.00
MOVJ C00512 BC00512 VJ=30.00
MOVJ C00513 BC00513 VJ=10.00
'**********************
'W53A
'**********************
SFTON P0306
MOVL C00514 BC00514 V=250.0
MOVL C00515 BC00515 V=83.3 PL=0
SFTOF
MACRO1 MJ#(0) ARGF10
ARCON
SFTON P0305
MOVL C00516 BC00516 V=10.8
ARCOF
SFTOF
MOVL C00517 BC00517 V=250.0
MOVJ C00518 BC00518 VJ=30.00
MOVJ C00519 BC00519 VJ=30.00
MOVJ C00520 BC00520 VJ=30.00
MOVJ C00521 BC00521 VJ=30.00
MOVJ C00522 BC00522 VJ=30.00
MOVJ C00523 BC00523 VJ=30.00
MOVL C00524 BC00524 V=250.0
'**********************
'W53B
'**********************
SFTON P0355
MOVL C00525 BC00525 V=250.0
MOVL C00526 BC00526 V=83.3 PL=0
SFTOF
MACRO1 MJ#(0) ARGF10
ARCON
SFTON P0356
MOVL C00527 BC00527 V=10.8
ARCOF
SFTOF
MOVL C00528 BC00528 V=333.3
MOVJ C00529 BC00529 VJ=30.00
MOVJ C00530 BC00530 VJ=30.00
MOVJ C00531 BC00531 VJ=30.00
MOVJ C00532 BC00532 VJ=30.00
MOVJ C00533 BC00533 VJ=30.00
'**********************
'W54A
'**********************
SFTON P0302
MOVL C00534 BC00534 V=250.0
MOVL C00535 BC00535 V=83.3 PL=0
SFTOF
MACRO1 MJ#(0) ARGF10
ARCON
SFTON P0301
MOVL C00536 BC00536 V=10.8
ARCOF
SFTOF
MOVL C00537 BC00537 V=333.3
MOVJ C00538 BC00538 VJ=20.00
MOVJ C00539 BC00539 VJ=30.00
MOVJ C00540 BC00540 VJ=30.00
MOVJ C00541 BC00541 VJ=30.00
MOVJ C00542 BC00542 VJ=30.00
'**********************
'W54B
'**********************
SFTON P0359
MOVL C00543 BC00543 V=250.0
MOVL C00544 BC00544 V=83.3 PL=0
SFTOF
MACRO1 MJ#(0) ARGF10
ARCON
SFTON P0360
MOVL C00545 BC00545 V=10.8
ARCOF
MOVL C00546 BC00546 V=333.3
SFTOF
MOVJ C00547 BC00547 VJ=30.00
MOVJ C00548 BC00548 VJ=30.00
MOVJ C00549 BC00549 VJ=30.00
MOVJ C00550 BC00550 VJ=40.00
MOVJ C00551 BC00551 VJ=40.00
MOVJ C00552 BC00552 VJ=10.00
MOVJ C00553 BC00553 VJ=10.00
MOVJ C00554 BC00554 VJ=10.00
MOVJ C00555 BC00555 VJ=15.00
MOVJ C00556 BC00556 VJ=15.00
MOVJ C00557 BC00557 VJ=15.00
MOVJ C00558 BC00558 VJ=15.00
'**********************
'W55A
'**********************
SFTON P0311
MOVL C00559 BC00559 V=166.7 PL=0
SFTOF
MACRO1 MJ#(0) ARGF10
ARCON
SFTON P0312
MOVL C00560 BC00560 V=10.8
MOVL C00561 BC00561 V=10.8
ARCOF
SFTOF
MOVL C00562 BC00562 V=150.0
MOVJ C00563 BC00563 VJ=10.00
MOVJ C00564 BC00564 VJ=10.00
MOVJ C00565 BC00565 VJ=10.00
MOVJ C00566 BC00566 VJ=10.00
MOVJ C00567 BC00567 VJ=10.00
MOVJ C00568 BC00568 VJ=10.00
MOVJ C00569 BC00569 VJ=30.00
MOVJ C00570 BC00570 VJ=30.00
MOVJ C00571 BC00571 VJ=20.00
MOVJ C00572 BC00572 VJ=30.00
MOVJ C00573 BC00573 VJ=20.00
MOVJ C00574 BC00574 VJ=20.00
MOVJ C00575 BC00575 VJ=30.00
MOVJ C00576 BC00576 VJ=20.00
MOVJ C00577 BC00577 VJ=20.00
'**********************
'W55B
'**********************
SFTON P0350
MOVL C00578 BC00578 V=333.3
MOVL C00579 BC00579 V=166.7 PL=0
SFTOF
MACRO1 MJ#(0) ARGF10
ARCON
SFTON P0349
MOVL C00580 BC00580 V=10.8
MOVL C00581 BC00581 V=10.8
ARCOF
SFTOF
MOVL C00582 BC00582 V=66.7
MOVJ C00583 BC00583 VJ=10.00
MOVJ C00584 BC00584 VJ=20.00
MOVJ C00585 BC00585 VJ=20.00
MOVJ C00586 BC00586 VJ=20.00
MOVJ C00587 BC00587 VJ=30.00
MOVJ C00588 BC00588 VJ=50.00
MOVJ C00589 BC00589 VJ=50.00
MOVJ C00590 BC00590 VJ=40.00
MOVJ C00591 BC00591 VJ=20.00
'**********************
'W56A
'**********************
SFTON P0308
MOVL C00592 BC00592 V=333.3
MOVL C00593 BC00593 V=166.7 PL=0
SFTOF
MACRO1 MJ#(0) ARGF10
ARCON
SFTON P0307
MOVL C00594 BC00594 V=10.8
ARCOF
SFTOF
MOVL C00595 BC00595 V=333.3
MOVJ C00596 BC00596 VJ=20.00
MOVJ C00597 BC00597 VJ=30.00
MOVJ C00598 BC00598 VJ=30.00
MOVJ C00599 BC00599 VJ=30.00
'**********************
'W56B
'**********************
SFTON P0353
MOVL C00600 BC00600 V=250.0
MOVL C00601 BC00601 V=166.7 PL=0
SFTOF
MACRO1 MJ#(0) ARGF10
ARCON
SFTON P0354
MOVL C00602 BC00602 V=10.8
ARCOF
SFTOF
MOVL C00603 BC00603 V=333.3
MOVJ C00604 BC00604 VJ=30.00
MOVJ C00605 BC00605 VJ=30.00
MOVJ C00606 BC00606 VJ=30.00
CALL JOB:MOVE_OUT_OF_TUNNEL
END
